// Se o estado de redundância deste PLC alterou...
IF NonRedData.bRedStateChanged THEN
	// Torna as saídas diferentes das entradas, garantindo que as consistências de dados
	// sejam feitas a partir de valores decorrentes de novas comunicações
	ATs.awModbus3HoldingWrite[0]:= ATs.awModbus3InputRegRead[0] + 100;
	// Inicializa temporizador para atrasar a consistência dos valores lidos, pois quando
	// o PLC assume como ativo, vai levar algum tempo até a comunicação ser estabelecida
	liAnalogTimer:= - ProjectConstants.iTimeToSkipAsActive;
ELSE
	// Se o protocolo MODBUS está rodando e se os dados são consistentes...
	IF DG_MODBUS_Client_3.tDiag.bRunning AND bStatusHolding AND bStatusInputReg THEN
		// Incrementa o valor escrito nos holding registers
		ATs.awModbus3HoldingWrite[0]:= ATs.awModbus3HoldingWrite[0] + 100;
		// Reseta o temporizador
		liAnalogTimer:= 0;
	ELSE
		// Acumula o tempo que passou
		liAnalogTimer:= liAnalogTimer + ProjectConstants.iMainTaskInterval;
		// Registra o tempo máximo
		MinMaxTimes.liAnaMaxTime_CheckModbus3:= MAX(MinMaxTimes.liAnaMaxTime_CheckModbus3, liAnalogTimer);
		// Caso o tempo máximo tenha sido extrapolado...
		IF liAnalogTimer >= ProjectConstants.iModbus3ReadWriteDelay THEN
			// Restarta o MODBUS caso o bug 17184 se manifeste.
			IF DG_MODBUS_Server_3.tStat.wActiveConnections = 0 THEN
				///DG_MODBUS_Server_3.tCommand.bRestart:= TRUE;
				PersistentVars.iBug17184_Counter_MDBUS3:= PersistentVars.iBug17184_Counter_MDBUS3 + 1;
				///iAnalogTimer:= - ProjectConstants.iTimeToSkipAsActive;
			ELSE	
				// Registra falha nos holding register, caso tenha ocorrido
				IF bStatusHolding = FALSE THEN
					PersistentVars.bModbus3ErrorHolding:= TRUE;
					awHoldingError_DataWr:= ATs.awModbus3HoldingWrite;
					awHoldingError_DataRd:= ATs.awModbus3HoldingRead;
				END_IF
				// Registra falha nos input register, caso tenha ocorrido
				IF bStatusInputReg = FALSE THEN
					PersistentVars.bModbus3ErrorInputReg:= TRUE;
					awInputRegError_DataWr:= ATs.awModbus3HoldingWrite;
					awInputRegError_DataRd:= ATs.awModbus3InputRegRead;
				END_IF
			END_IF
		END_IF
	END_IF
END_IF

// Atualiza os valores escritos
FOR wIndex:= 1 TO 119 BY 1 DO
	ATs.awModbus3HoldingWrite[wIndex]:= ATs.awModbus3HoldingWrite[wIndex - 1] + wIndex;
END_FOR

//
// Calcula a taxa média de comunicação
//

// Incrementa o número de milisegundos que transcorreram
iMilisecondsCounter:= iMilisecondsCounter + ProjectConstants.iMainTaskInterval;
// Se já se passou o tempo configurado desde a última média realizada...
IF iMilisecondsCounter >= ProjectConstants.iMsToComputeComRate THEN
	// Só calcula se o contador não virou
	IF DG_MODBUS_Client_3.tStat.wRXNormalResponses > wOldRXNormalResponses THEN
		// Calcula a taxa de comunicação atual
		MinMaxTimes.diModbus3BytesPerSec:=	WORD_TO_DINT(DG_MODBUS_Client_3.tStat.wRXNormalResponses - wOldRXNormalResponses) *
											iBytesPerResponse * 1000 / iMilisecondsCounter;
	END_IF
	// Zera o número de milisegundos transcorridos
	iMilisecondsCounter:= 0;
	// Salva número de respostas atuais
	wOldRXNormalResponses:= DG_MODBUS_Client_3.tStat.wRXNormalResponses;
END_IF

// Registra o tempo do sistema
SysTimeGetUs(uliPouEndTime);
// Calcula duração mínima/máxima desta POU
MinMaxTimes.uliPouMinTime_CheckModbus3:= MIN(MinMaxTimes.uliPouMinTime_CheckModbus3, uliPouEndTime - uliPouIniTime);
MinMaxTimes.uliPouMaxTime_CheckModbus3:= MAX(MinMaxTimes.uliPouMaxTime_CheckModbus3, uliPouEndTime - uliPouIniTime);

END_PROGRAM

// Device/Application/UserPOUs/Non-Redundant/CheckModbus4
PROGRAM CheckModbus4
VAR
	wIndex : WORD;
	bStatusCoil : BOOL;
	bStatusStatus : BOOL;
	bStatusHolding : BOOL;
	bStatusInputReg : BOOL;
	liDigitalTimer : LINT := 0;
	liAnalogTimer : LINT := 0;
	abCoilsError_DataWr : ARRAY [0..1919] OF BOOL;
	abCoilsError_DataRd : ARRAY [0..1919] OF BOOL;
	abStatusError_DataWr : ARRAY [0..1919] OF BOOL;
	abStatusError_DataRd : ARRAY [0..1919] OF BOOL;
	awHoldingError_DataWr : ARRAY [0..119] OF WORD;
	awHoldingError_DataRd : ARRAY [0..119] OF WORD;
	awInputRegError_DataWr : ARRAY [0..119] OF WORD;
	awInputRegError_DataRd : ARRAY [0..119] OF WORD;
	wOldRXNormalResponses : WORD;
	iMilisecondsCounter : INT;
	iBytesPerResponse : INT := 240;
	uliPouIniTime : ULINT;
	uliPouEndTime : ULINT;
END_VAR

// Consistencia da integridade dos dados trocados via MODBUS

// Registra o tempo do sistema
SysTimeGetUs(uliPouIniTime);

//
// Controle e consistência dos coils e input status
//

// Consiste os valores lidos
bStatusCoil:= TRUE;
bStatusStatus:= TRUE;
FOR wIndex:= 0 TO 1919 BY 1 DO
	bStatusCoil:= bStatusCoil AND (ModbusSymbol.abModbus4CoilsRead[wIndex] = ModbusSymbol.abModbus4CoilsWrite[wIndex]);
	bStatusStatus:= bStatusStatus AND (ModbusSymbol.abModbus4StatusRead[wIndex] = ModbusSymbol.abModbus4CoilsWrite[wIndex]);
END_FOR

// Se o estado de redundância deste PLC alterou...
IF NonRedData.bRedStateChanged THEN
	// Torna as saídas diferentes das entradas, garantindo que as consistências de dados
	// sejam feitas a partir de valores decorrentes de novas comunicações
	ModbusSymbol.abModbus4CoilsWrite[0]:= NOT ModbusSymbol.abModbus4StatusRead[0];
	// Inicializa temporizador para atrasar a consistência dos valores lidos, pois quando
	// o PLC assume como ativo, vai levar algum tempo até a comunicação ser estabelecida
	liDigitalTimer:= - ProjectConstants.iTimeToSkipAsActive;
ELSE
	// Se o protocolo MODBUS está rodando e se os dados são consistentes...
	IF DG_MODBUS_Client_4.tDiag.bRunning AND bStatusCoil AND bStatusStatus THEN
		// Complementa o valor dos coils
		ModbusSymbol.abModbus4CoilsWrite[0]:= NOT ModbusSymbol.abModbus4CoilsWrite[0];
		// Reseta o temporizador
		liDigitalTimer:= 0;
	ELSE
		// Acumula o tempo que passou
		liDigitalTimer:= liDigitalTimer + ProjectConstants.iMainTaskInterval;
		// Registra o tempo máximo
		MinMaxTimes.liDigMaxTime_CheckModbus4:= MAX(MinMaxTimes.liDigMaxTime_CheckModbus4, liDigitalTimer);
		// Caso o tempo máximo tenha sido extrapolado...
		IF liDigitalTimer >= ProjectConstants.iModbus4ReadWriteDelay THEN
		// Restarta o MODBUS caso o bug 17184 se manifeste.
			IF DG_MODBUS_Server_4.tStat.wActiveConnections = 0 THEN
				///DG_MODBUS_Server_4.tCommand.bRestart:= TRUE;
				PersistentVars.iBug17184_CounterDig_MDBUS4:= PersistentVars.iBug17184_CounterDig_MDBUS4 + 1;
				///iDigitalTimer:= - ProjectConstants.iTimeToSkipAsActive;
			ELSE
				// Registra falha nos coils, caso tenha ocorrido
				IF bStatusCoil = FALSE THEN
					PersistentVars.bModbus4ErrorCoil:= TRUE;
					abCoilsError_DataWr:= ModbusSymbol.abModbus4CoilsWrite;
					abCoilsError_DataRd:= ModbusSymbol.abModbus4CoilsRead;
				END_IF
				// Registra falha nos inputs, caso tenha ocorrido
				IF bStatusStatus = FALSE THEN
					PersistentVars.bModbus4ErrorStatus:= TRUE;
					abStatusError_DataWr:= ModbusSymbol.abModbus4CoilsWrite;
					abStatusError_DataRd:= ModbusSymbol.abModbus4StatusRead;
				END_IF
			END_IF
		END_IF
	END_IF
END_IF

// Atualiza os valores escritos
FOR wIndex:= 1 TO 1919 BY 1 DO
	ModbusSymbol.abModbus4CoilsWrite[wIndex]:= NOT ModbusSymbol.abModbus4CoilsWrite[wIndex - 1];
END_FOR

//
// Controle e consistência dos holding registers
//

// Consiste os valores lidos
bStatusHolding:= TRUE;
bStatusInputReg:= TRUE;
FOR wIndex:= 0 TO 119 BY 1 DO
	bStatusHolding:= bStatusHolding AND (ModbusSymbol.awModbus4HoldingRead[wIndex] = ModbusSymbol.awModbus4HoldingWrite[wIndex]);
	bStatusInputReg:= bStatusInputReg AND (ModbusSymbol.awModbus4InputRegRead[wIndex] = ModbusSymbol.awModbus4HoldingWrite[wIndex]);
END_FOR

// Se o estado de redundância deste PLC alterou...
IF NonRedData.bRedStateChanged THEN
	// Torna as saídas diferentes das entradas, garantindo que as consistências de dados
	// sejam feitas a partir de valores decorrentes de novas comunicações
	ModbusSymbol.awModbus4HoldingWrite[0]:= ModbusSymbol.awModbus4InputRegRead[0] + 100;
	// Inicializa temporizador para atrasar a consistência dos valores lidos, pois quando
	// o PLC assume como ativo, vai levar algum tempo até a comunicação ser estabelecida
	liAnalogTimer:= - ProjectConstants.iTimeToSkipAsActive;
ELSE
	// Se o protocolo MODBUS está rodando e se os dados são consistentes...
	IF DG_MODBUS_Client_4.tDiag.bRunning AND bStatusHolding AND bStatusInputReg THEN
		// Incrementa o valor escrito nos holding registers
		ModbusSymbol.awModbus4HoldingWrite[0]:= ModbusSymbol.awModbus4HoldingWrite[0] + 100;
		// Reseta o temporizador
		liAnalogTimer:= 0;
	ELSE
		// Acumula o tempo que passou
		liAnalogTimer:= liAnalogTimer + ProjectConstants.iMainTaskInterval;
		// Registra o tempo máximo
		MinMaxTimes.liAnaMaxTime_CheckModbus4:= MAX(MinMaxTimes.liAnaMaxTime_CheckModbus4, liAnalogTimer);
		// Caso o tempo máximo tenha sido extrapolado...
		IF liAnalogTimer >= ProjectConstants.iModbus4ReadWriteDelay THEN
			// Restarta o MODBUS caso o bug 17184 se manifeste.
			IF DG_MODBUS_Server_4.tStat.wActiveConnections = 0 THEN
				///DG_MODBUS_Server_4.tCommand.bRestart:= TRUE;
				PersistentVars.iBug17184_Counter_MDBUS4:= PersistentVars.iBug17184_Counter_MDBUS4 + 1;
				///AnalogTimer:= - ProjectConstants.iTimeToSkipAsActive;
			ELSE
				// Registra falha nos holding register, caso tenha ocorrido
				IF bStatusHolding = FALSE THEN
					PersistentVars.bModbus4ErrorHolding:= TRUE;
					awHoldingError_DataWr:= ModbusSymbol.awModbus4HoldingWrite;
					awHoldingError_DataRd:= ModbusSymbol.awModbus4HoldingRead;
				END_IF
				// Registra falha nos input register, caso tenha ocorrido
				IF bStatusInputReg = FALSE THEN
					PersistentVars.bModbus4ErrorInputReg:= TRUE;
					awInputRegError_DataWr:= ModbusSymbol.awModbus4HoldingWrite;
					awInputRegError_DataRd:= ModbusSymbol.awModbus4InputRegRead;
				END_IF
			END_IF
		END_IF
	END_IF
END_IF

// Atualiza os valores escritos
FOR wIndex:= 1 TO 119 BY 1 DO
	ModbusSymbol.awModbus4HoldingWrite[wIndex]:= ModbusSymbol.awModbus4HoldingWrite[wIndex - 1] + wIndex;
END_FOR

//
// Calcula a taxa média de comunicação
//

// Incrementa o número de milisegundos que transcorreram
iMilisecondsCounter:= iMilisecondsCounter + ProjectConstants.iMainTaskInterval;
// Se já se passou o tempo configurado desde a última média realizada...
IF iMilisecondsCounter >= ProjectConstants.iMsToComputeComRate THEN
	// Só calcula se o contador não virou
	IF DG_MODBUS_Client_4.tStat.wRXNormalResponses > wOldRXNormalResponses THEN
		// Calcula a taxa de comunicação atual
		MinMaxTimes.diModbus4BytesPerSec:=	WORD_TO_DINT(DG_MODBUS_Client_4.tStat.wRXNormalResponses - wOldRXNormalResponses) *
											iBytesPerResponse * 1000 / iMilisecondsCounter;
	END_IF
	// Zera o número de milisegundos transcorridos
	iMilisecondsCounter:= 0;
	// Salva número de respostas atuais
	wOldRXNormalResponses:= DG_MODBUS_Client_4.tStat.wRXNormalResponses;
END_IF

// Registra o tempo do sistema
SysTimeGetUs(uliPouEndTime);
// Calcula duração mínima/máxima desta POU
MinMaxTimes.uliPouMinTime_CheckModbus4:= MIN(MinMaxTimes.uliPouMinTime_CheckModbus4, uliPouEndTime - uliPouIniTime);
MinMaxTimes.uliPouMaxTime_CheckModbus4:= MAX(MinMaxTimes.uliPouMaxTime_CheckModbus4, uliPouEndTime - uliPouIniTime);

END_PROGRAM

// Device/Application/UserPOUs/Redundant/CheckProfibusIOs
PROGRAM CheckProfibusIOs
VAR
	iAnalogHigh : INT := 30000;
	iAnalogLow : INT := 1500;
	iAnalogError : INT := 100;
	iAnalogStep : INT := 1500;
	abErrorLoopBack : ARRAY [0..3] OF BYTE;
	uliPouIniTime : ULINT;
	uliPouEndTime : ULINT;
END_VAR

// Registra o tempo do sistema
SysTimeGetUs(uliPouIniTime);

// Zera variáveis em caso de comando para reinicializar os contadores de diagnóstico
	IF Symbolics.bEnableCleanStats_CheckProfibusIOs = TRUE THEN
		abErrorLoopBack[0]:= 0;
		abErrorLoopBack[1]:= 0;
		abErrorLoopBack[2]:= 0;
		abErrorLoopBack[3]:= 0;
		Symbolics.bEnableCleanStats_CheckProfibusIOs:= FALSE;
	END_IF



//
// Teste de consistência de I/Os PROFIBUS digitais e analógicos ligados ao PO5065.
//

// Se o mestre Profibus está presente no barramento e se a primeira cabeça (endereço 5) está ativa na rede...
IF (((DG_NX3030.tDetailed.WHSB.adwModulePresenceStatus[0] AND 2#001000000) > 0) AND
	 (DG_NX5001_1.tRedund.tActivNtw.bSlave_5 = TRUE)) OR
   (((DG_NX3030.tDetailed.WHSB.adwModulePresenceStatus[0] AND 2#100000000) > 0) AND
	 (DG_NX5001_2.tRedund.tActivNtw.bSlave_5 = TRUE)) THEN
	// Se os módulos de entrada e de saída digital estiverem presentes no barramento...
	IF (DG_PO5065_05.tPbusHeadA.tModule_0to7_Status.bModuleNotFound_00 = FALSE) AND
	   (DG_PO5065_05.tPbusHeadA.tModule_0to7_Status.bModuleNotFound_01 = FALSE) AND
	   (DG_PO5065_05.tPbusHeadB.tModule_0to7_Status.bModuleNotFound_00 = FALSE) AND 
	   (DG_PO5065_05.tPbusHeadB.tModule_0to7_Status.bModuleNotFound_01 = FALSE) THEN
		// Consiste entradas e saídas digitais, interligadas fisicamente
		IF REM05_PO2020_G0 = REM05_PO1000_G0 THEN
			// Incrementa o estado das saídas digitais
			REM05_PO2020_G0:= REM05_PO2020_G0 + 1;
			// Reseta o temporizador
			NonRedData.iProfibus5DigTimer:= 0;
		ELSE
			// Acumula o tempo que passou
			NonRedData.iProfibus5DigTimer:= NonRedData.iProfibus5DigTimer + ProjectConstants.iMainTaskInterval;
			// Registra o tempo máximo
			MinMaxTimes.liDigMaxTime_CheckProfibusIOs:= MAX(MinMaxTimes.liDigMaxTime_CheckProfibusIOs, NonRedData.iProfibus5DigTimer);
			// Aguarda a passagem do tempo antes de considerar falha
			IF NonRedData.iProfibus5DigTimer = ProjectConstants.iProfibusDelayDigital THEN
				// Contabiliza erro de consistência dos pontos digitais
				PersistentVars.dwSlave5DigIOsErrors:= PersistentVars.dwSlave5DigIOsErrors + 1;
				//Armazena o erro da entrada e saida
				abErrorLoopBack[0]:= REM05_PO1000_G0;
				abErrorLoopBack[1]:= REM05_PO2020_G0;
			ELSE
				//Gabriel Fonseca - 28/10/2022
				//Verifica se congelou por mais de um ciclo, retornar >= no if acima 
				IF NonRedData.iProfibus5DigTimer >= 2* ProjectConstants.iProfibusDelayDigital THEN
					PersistentVars.bFrozenErrorRem05TORem05:= TRUE;
				END_IF
			END_IF
		END_IF
	// Se algum dos módulos de entrada e de saída digital estiverem ausentes do barramento...
	ELSE
		// Acumula o tempo que passou
		NonRedData.iProfibus5DigTimer:= NonRedData.iProfibus5DigTimer + ProjectConstants.iMainTaskInterval;
		// Registra o tempo máximo
		MinMaxTimes.liDigMaxTime_CheckProfibusIOs:= MAX(MinMaxTimes.liDigMaxTime_CheckProfibusIOs, NonRedData.iProfibus5DigTimer);
		// Aguarda a passagem do tempo antes de considerar falha
		IF NonRedData.iProfibus5DigTimer >= ProjectConstants.iProfibusDelayDigital THEN
			// Contabiliza erro de módulo ausente do barramento
			PersistentVars.dwSlave5ModulesOut:= PersistentVars.dwSlave5ModulesOut + 1;
		END_IF
	END_IF
// Se o mestre Profibus está ausente do barramento ou se a primeira cabeça (endereço 5) não está ativa na rede...
ELSE
	// Acumula o tempo que passou
	NonRedData.iProfibus5DigTimer:= NonRedData.iProfibus5DigTimer + ProjectConstants.iMainTaskInterval;
	// Registra o tempo máximo
	MinMaxTimes.liDigMaxTime_CheckProfibusIOs:= MAX(MinMaxTimes.liDigMaxTime_CheckProfibusIOs, NonRedData.iProfibus5DigTimer);
	// Aguarda a passagem do tempo antes de considerar falha
	IF NonRedData.iProfibus5DigTimer >= ProjectConstants.iProfibusDelayDigital THEN
		// Contabiliza erro de Cabeça não ativa na rede
		PersistentVars.dwSlave5Unavailable:= PersistentVars.dwSlave5Unavailable + 1;
	END_IF
END_IF

// Se o mestre Profibus está presente no barramento e se a segunda cabeça (endereço 10) está ativa na rede...
IF (((DG_NX3030.tDetailed.WHSB.adwModulePresenceStatus[0] AND 2#001000000) > 0) AND 
	 (DG_NX5001_1.tRedund.tActivNtw.bSlave_10 = TRUE)) OR
   (((DG_NX3030.tDetailed.WHSB.adwModulePresenceStatus[0] AND 2#100000000) > 0) AND 
	 (DG_NX5001_2.tRedund.tActivNtw.bSlave_10 = TRUE)) THEN
	// Se os módulos de entrada e de saída analógica estiverem presentes no barramento...
	IF (DG_PO5065_10.tPbusHeadA.tModule_0to7_Status.bModuleNotFound_00 = FALSE) AND
	   (DG_PO5065_10.tPbusHeadA.tModule_0to7_Status.bModuleNotFound_01 = FALSE) AND
	   (DG_PO5065_10.tPbusHeadB.tModule_0to7_Status.bModuleNotFound_00 = FALSE) AND
	   (DG_PO5065_10.tPbusHeadB.tModule_0to7_Status.bModuleNotFound_01 = FALSE) THEN
		// Consistência da primeira entrada analógica (rampa)
		IF (WORD_TO_INT(REM10_PO1212_C00) >= (Symbolics.iAnalogValue - iAnalogError)) AND
		   (WORD_TO_INT(REM10_PO1212_C00) <= (Symbolics.iAnalogValue + iAnalogError)) THEN
			// Implementa rampa analógica
			Symbolics.iAnalogValue:= Symbolics.iAnalogValue + iAnalogStep;
			// Ajusta subida/descida da rampa analógica
			IF Symbolics.iAnalogValue >= iAnalogHigh THEN
				Symbolics.iAnalogValue:= iAnalogHigh;
				iAnalogStep:= -iAnalogStep;
			END_IF
			IF Symbolics.iAnalogValue <= iAnalogLow	THEN
				Symbolics.iAnalogValue:= iAnalogLow;
				iAnalogStep:= -iAnalogStep;
			END_IF
			// Primeira saída analógica é uma rampa
			REM10_PO2132_C00:= INT_TO_WORD(Symbolics.iAnalogValue);
			// Reseta o temporizador
			NonRedData.iProfibus10AnaTimer:= 0;
		ELSE
			// Acumula o tempo que passou
			NonRedData.iProfibus10AnaTimer:= NonRedData.iProfibus10AnaTimer + ProjectConstants.iMainTaskInterval;
			// Registra o tempo máximo
			MinMaxTimes.liAnaMaxTime_CheckProfibusIOs:= MAX(MinMaxTimes.liAnaMaxTime_CheckProfibusIOs, NonRedData.iProfibus10AnaTimer);
			// Aguarda a passagem do tempo antes de considerar falha
			IF NonRedData.iProfibus10AnaTimer >= ProjectConstants.iProfibusDelayAnalog THEN
				// Contabiliza erro de consistência dos pontos analógicos
				PersistentVars.dwSlave10AnaIOsErrors:= PersistentVars.dwSlave10AnaIOsErrors + 1;
				// Salva os valores errados
				PersistentVars.wErrorValuePO2132C00:= REM10_PO2132_C00;
				PersistentVars.wErrorValuePO1212C00:= REM10_PO1212_C00;
			END_IF
		END_IF
	// Se algum dos módulos de entrada e de saída analógica estiverem ausentes do barramento...
	ELSE
		// Acumula o tempo que passou
		NonRedData.iProfibus10AnaTimer:= NonRedData.iProfibus10AnaTimer + ProjectConstants.iMainTaskInterval;
		// Registra o tempo máximo
		MinMaxTimes.liAnaMaxTime_CheckProfibusIOs:= MAX(MinMaxTimes.liAnaMaxTime_CheckProfibusIOs, NonRedData.iProfibus10AnaTimer);
		// Aguarda a passagem do tempo antes de considerar falha
		IF NonRedData.iProfibus10AnaTimer >= ProjectConstants.iProfibusDelayAnalog THEN
			// Contabiliza erro de módulo ausente do barramento
			PersistentVars.dwSlave10ModulesOut:= PersistentVars.dwSlave10ModulesOut + 1;
		END_IF
	END_IF
// Se o mestre Profibus está ausente do barramento ou se a segunda cabeça (endereço 10) não está ativa na rede...
ELSE
	// Acumula o tempo que passou
	NonRedData.iProfibus10AnaTimer:= NonRedData.iProfibus10AnaTimer + ProjectConstants.iMainTaskInterval;
	// Registra o tempo máximo
	MinMaxTimes.liAnaMaxTime_CheckProfibusIOs:= MAX(MinMaxTimes.liAnaMaxTime_CheckProfibusIOs, NonRedData.iProfibus10AnaTimer);
	// Aguarda a passagem do tempo antes de considerar falha
	IF NonRedData.iProfibus10AnaTimer >= ProjectConstants.iProfibusDelayAnalog THEN
		// Contabiliza erro de Cabeça não ativa na rede
		PersistentVars.dwSlave10Unavailable:= PersistentVars.dwSlave10Unavailable + 1;
	END_IF
END_IF

//
// Teste de consistência de I/Os PROFIBUS digital ligado ao PO5063.
//

// Se o mestre Profibus está presente no barramento e se a cabeça (endereço 3) está ativa na rede...
IF (((DG_NX3030.tDetailed.WHSB.adwModulePresenceStatus[0] AND 2#10000000000000000) > 0) AND //posição 16
	 (DG_NX5001_3.tMstStatus.abySlv_State.bSlave_4 = TRUE)) THEN
	// Se o módulo de entrada digital estiver presente no barramento...
	IF DG_PO5063_04.tPbusHeadA.tModule_0to7_Status.bModuleNotFound_00 = FALSE THEN
		// Consiste entradas e saídas digitais, interligadas fisicamente
		
		IF REM05_PO2020_G1 = REM04_PO1000_G0 THEN
			// Incrementa o estado das saídas digitais
			REM05_PO2020_G1:= REM05_PO2020_G1 + 1;
			// Reseta o temporizador
			NonRedData.iProfibus3DigTimer:= 0;
		ELSE
			// Acumula o tempo que passou
			NonRedData.iProfibus3DigTimer:= NonRedData.iProfibus3DigTimer + ProjectConstants.iMainTaskInterval;
			// Registra o tempo máximo
			MinMaxTimes.liDigMaxTime_CheckProfibusIOs:= MAX(MinMaxTimes.liDigMaxTime_CheckProfibusIOs, NonRedData.iProfibus3DigTimer);
			// Aguarda a passagem do tempo antes de considerar falha
			IF NonRedData.iProfibus3DigTimer = ProjectConstants.iProfibusDelayDigital THEN
				// Contabiliza erro de consistência dos pontos digitais
				PersistentVars.dwSlave3DigIOsErrors:= PersistentVars.dwSlave3DigIOsErrors + 1;
				//Armazena o erro da entrada e saida
				abErrorLoopBack[2] := REM04_PO1000_G0;
				abErrorLoopBack[3] := REM05_PO2020_G1;
			ELSE 
				//Gabriel Fonseca - 28/10/2022
				//Verifica se congelou por mais de um ciclo, retornar >= no if acima 
				IF NonRedData.iProfibus3DigTimer >= 2* ProjectConstants.iProfibusDelayDigital THEN
					PersistentVars.bFrozenErrorRem05TORem04:= TRUE;
				END_IF
			END_IF
			
		END_IF
	// Se o módulo de entrada digital estiver ausente do barramento...
	ELSE
		// Acumula o tempo que passou
		NonRedData.iProfibus3DigTimer:= NonRedData.iProfibus3DigTimer + ProjectConstants.iMainTaskInterval;
		// Registra o tempo máximo
		MinMaxTimes.liDigMaxTime_CheckProfibusIOs:= MAX(MinMaxTimes.liDigMaxTime_CheckProfibusIOs, NonRedData.iProfibus3DigTimer);
		// Aguarda a passagem do tempo antes de considerar falha
		IF NonRedData.iProfibus3DigTimer >= ProjectConstants.iProfibusDelayDigital THEN
			// Contabiliza erro de módulo ausente do barramento
			PersistentVars.dwSlave3ModulesOut:= PersistentVars.dwSlave3ModulesOut + 1;
		END_IF
	END_IF
// Se o mestre Profibus está ausente do barramento ou se a cabeça (endereço 3) não está ativa na rede...
ELSE
	// Acumula o tempo que passou
	NonRedData.iProfibus3DigTimer:= NonRedData.iProfibus3DigTimer + ProjectConstants.iMainTaskInterval;
	// Registra o tempo máximo
	MinMaxTimes.liDigMaxTime_CheckProfibusIOs:= MAX(MinMaxTimes.liDigMaxTime_CheckProfibusIOs, NonRedData.iProfibus3DigTimer);
	// Aguarda a passagem do tempo antes de considerar falha
	IF NonRedData.iProfibus3DigTimer >= ProjectConstants.iProfibusDelayDigital THEN
		// Contabiliza erro de Cabeça não ativa na rede
		PersistentVars.dwSlave3Unavailable:= PersistentVars.dwSlave3Unavailable + 1;
	END_IF
END_IF

//*****************************************************************************************************************************************************************************
//
// Teste de consistência de I/Os PROFIBUS ligados a remotas Nexto

// Registra o tempo do sistema
SysTimeGetUs(uliPouEndTime);
// Calcula duração mínima/máxima desta POU
MinMaxTimes.uliPouMinTime_CheckProfibusIOs:= MIN(MinMaxTimes.uliPouMinTime_CheckProfibusIOs, uliPouEndTime - uliPouIniTime);
MinMaxTimes.uliPouMaxTime_CheckProfibusIOs:= MAX(MinMaxTimes.uliPouMaxTime_CheckProfibusIOs, uliPouEndTime - uliPouIniTime);

END_PROGRAM

// Device/Application/UserPOUs/Redundant/CheckRecipe
PROGRAM CheckRecipe
VAR
	sName : STRING := 'ReceitaMinima';
	sDef : STRING := 'Machine01';
	mRET : RECIPE_RETURN_VALUES;
	boolStartProcess : BOOL;
	bTestRecipe : BOOL;
	iCounterCycle : INT;
	bOneCycle : BOOL;
	uliPouIniTime : ULINT;
	uliPouEndTime : ULINT;
END_VAR

//*****************************************************************************
// Autor(es): Roberto Martiny
// Descrição:
// Esta POU testa a funcionalidade do Recipe Manager.
//*****************************************************************************

// Registra o tempo do sistema
SysTimeGetUs(uliPouIniTime);

//*****************************************************************************
// Testa Recipe Manager

IF bOneCycle = FALSE THEN
	mRET := WriteRecipe(SDef,SName);
	bOneCycle := TRUE;
END_IF

iCounterCycle := iCounterCycle+1;

IF bTestRecipe = FALSE AND iCounterCycle > 1 THEN
	IF Recipe.iRecipeValueA <> -1000 OR Recipe.iRecipeValueB <> 1 OR Recipe.iRecipeValueC <> -900 THEN
	PersistentVars.dwRecipeErrors := PersistentVars.dwRecipeErrors +1;
	END_IF
	// fica por 10 ciclos consistindo este recipe
	IF iCounterCycle > 10 THEN
		iCounterCycle :=0;
		bTestRecipe := TRUE;
		sName := 'ReceitaMaxima';
		mRET := WriteRecipe(SDef,SName);	
	END_IF	
END_IF

IF bTestRecipe = TRUE  AND iCounterCycle > 1 THEN
	IF Recipe.iRecipeValueA <> 1000 OR Recipe.iRecipeValueB <> 900 OR Recipe.iRecipeValueC <> -1 THEN
	PersistentVars.dwRecipeErrors := PersistentVars.dwRecipeErrors +1;
	END_IF
	// fica por 10 ciclos consistindo este recipe
	IF iCounterCycle > 10 THEN
		iCounterCycle :=0;
		bTestRecipe := FALSE;
		sName := 'ReceitaMinima';
		mRET := WriteRecipe(SDef,SName);
	END_IF	
END_IF

// Verifica retorno da função de escrita do Recipe
IF mRET <> RECIPE_RETURN_VALUES.ERROR_OK THEN
	PersistentVars.dwRecipeReturnError := mRET;
END_IF;
//*****************************************************************************

// Registra o tempo do sistema
SysTimeGetUs(uliPouEndTime);
// Calcula duração mínima/máxima desta POU
MinMaxTimes.uliPouMinTime_CheckRecipe:= MIN(MinMaxTimes.uliPouMinTime_CheckRecipe, uliPouEndTime - uliPouIniTime);
MinMaxTimes.uliPouMaxTime_CheckRecipe:= MAX(MinMaxTimes.uliPouMaxTime_CheckRecipe, uliPouEndTime - uliPouIniTime);

END_PROGRAM

// Device/Application/UserPOUs/Redundant/CheckSoe
PROGRAM CheckSoe
VAR
	wCounter : WORD := 0;
	wOldCounter : WORD := 0;
	// Memórias de salvamento dos erros
	wMemError_Soe1OverflowOldCounter : WORD;
	wMemError_Soe2OverflowOldCounter : WORD;
	wMemError_Soe1Diagnostic : WORD;
	wMemError_Soe1OldCounter : WORD;
	wMemError_Soe2Diagnostic : WORD;
	wMemError_Soe2OldCounter : WORD;
	uliPouIniTime : ULINT;
	uliPouEndTime : ULINT;
END_VAR

// Gera dois eventos SOE a cada ciclo nos dois servers e consiste a existência dos mesmos na fila.

// Registra o tempo do sistema
SysTimeGetUs(uliPouIniTime);

// Retorna se for o primeiro ciclo como ativo, pois os diagnósticos não estão atualizados
// Retorna também se for o segundo ciclo como ativo, devido ao BUG 17134
IF NonRedData.aeLastRedState[1] <> REDUNDANCY_STATE.ACTIVE OR
   NonRedData.aeLastRedState[2] <> REDUNDANCY_STATE.ACTIVE THEN
	RETURN;
END_IF

// Se for a primeira vez que esta POU será executada como PLC ativo, deve considerar a
// quantidade de eventos que já estão na fila, inclusive o overflow, pois são retentivos
IF NonRedData.bSoeFirstCheckCycle = TRUE THEN
	wCounter:= wOldCounter:= DG_NX3030.tDetailed.SOE[1].wEventsCounter +
							 2 * BOOL_TO_WORD(DG_NX3030.tDetailed.SOE[1].bOverflowStatus);
	NonRedData.bSoeFirstCheckCycle:= FALSE;
END_IF

//
// Consistência da indicação de overflow
//

// Se já ultrapassou o limite de eventos suportado, deve ter ligado o overflow
IF wOldCounter > ProjectConstants.wSoeEventQueueSize THEN
	// Se o flag de overflow da fila 1 está desligado...
	IF DG_NX3030.tDetailed.SOE[1].bOverflowStatus = FALSE THEN
		// Indica a ocorrência de um falso overflow
		PersistentVars.bSOE1FalseOverflow:= TRUE;
		// Salva os valores nas memórias de erro
		wMemError_Soe1OverflowOldCounter:= wOldCounter;
	END_IF
	// Se o flag de overflow da fila 2 está desligado...
	IF DG_NX3030.tDetailed.SOE[2].bOverflowStatus = FALSE THEN
		// Indica a ocorrência de um falso overflow
		PersistentVars.bSOE2FalseOverflow:= TRUE;
		// Salva os valores nas memórias de erro
		wMemError_Soe2OverflowOldCounter:= wOldCounter;
	END_IF
// Se não ultrapassou o limite de eventos suportado, não deve ter ligado o overflow
ELSE
	// Se o flag de overflow da fila 1 está ligado...
	IF DG_NX3030.tDetailed.SOE[1].bOverflowStatus = TRUE THEN
		// Indica a ocorrência de um falso overflow
		PersistentVars.bSOE1FalseOverflow:= TRUE;
		// Salva os valores nas memórias de erro
		wMemError_Soe1OverflowOldCounter:= wOldCounter;
	END_IF
	// Se o flag de overflow da fila 2 está ligado...
	IF DG_NX3030.tDetailed.SOE[2].bOverflowStatus = TRUE THEN
		// Indica a ocorrência de um falso overflow
		PersistentVars.bSOE2FalseOverflow:= TRUE;
		// Salva os valores nas memórias de erro
		wMemError_Soe2OverflowOldCounter:= wOldCounter;
	END_IF
END_IF

//
// Consistência da quantidade de eventos gerados
//

// Se não ultrapassou o limite de eventos suportado pela fila...
IF wOldCounter <= ProjectConstants.wSoeEventQueueSize THEN
	// Se o número de eventos na fila 1 não confere com o número de eventos gerados...
	IF DG_NX3030.tDetailed.SOE[1].wEventsCounter <> wOldCounter THEN
		// Indica falha na quantidade de eventos
		PersistentVars.bSOE1EventsMismatch:= TRUE;
		// Salva os valores nas memórias de erro
		wMemError_Soe1Diagnostic:= DG_NX3030.tDetailed.SOE[1].wEventsCounter;
		wMemError_Soe1OldCounter:= wOldCounter;
	END_IF
	// Se o número de eventos na fila 2 não confere com o número de eventos gerados...
	IF DG_NX3030.tDetailed.SOE[2].wEventsCounter <> wOldCounter THEN
		// Indica falha na quantidade de eventos
		PersistentVars.bSOE2EventsMismatch:= TRUE;
		// Salva os valores nas memórias de erro
		wMemError_Soe2Diagnostic:= DG_NX3030.tDetailed.SOE[2].wEventsCounter;
		wMemError_Soe2OldCounter:= wOldCounter;
	END_IF
// Se já ultrapassou o limite de eventos suportado pela fila...
ELSE
	// Se o número de eventos na fila 1 não confere com o número máximo...
	IF DG_NX3030.tDetailed.SOE[1].wEventsCounter <> ProjectConstants.wSoeEventQueueSize THEN
		// Indica falha na quantidade de eventos
		PersistentVars.bSOE1EventsMismatch:= TRUE;
		// Salva os valores nas memórias de erro
		wMemError_Soe1Diagnostic:= DG_NX3030.tDetailed.SOE[1].wEventsCounter;
		wMemError_Soe1OldCounter:= wOldCounter;
	END_IF
	// Se o número de eventos na fila 2 não confere com o número máximo...
	IF DG_NX3030.tDetailed.SOE[2].wEventsCounter <> ProjectConstants.wSoeEventQueueSize THEN
		// Indica falha na quantidade de eventos
		PersistentVars.bSOE2EventsMismatch:= TRUE;
		// Salva os valores nas memórias de erro
		wMemError_Soe2Diagnostic:= DG_NX3030.tDetailed.SOE[2].wEventsCounter;
		wMemError_Soe2OldCounter:= wOldCounter;
	END_IF
END_IF

// Salva o contador atual para consistir no próximo ciclo. Isto é necessário pois
// os diagnósticos (por exemplo, de eventos na fila) estão defasados em um ciclo:
// ao final da MainPrg, primeiro são gerados os diagnósticos e depois os eventos.  
wOldCounter:= wCounter;

// Enquanto não atingir o limite, gera mais dois eventos por ciclo
IF wCounter < ANY_TO_WORD(wCounter + 2) THEN
	ATs.bSOEPoint000:= NOT(ATs.bSOEPoint000);
	ATs.bSOEPoint999:= NOT(ATs.bSOEPoint999);
	wCounter:= wCounter + 2;
// Código para manter a instrução IF simétrica
ELSE
	ATs.bSOEPoint000:= ATs.bSOEPoint000;
	ATs.bSOEPoint999:= ATs.bSOEPoint999;
	wCounter:= wCounter + 0;
END_IF

// Registra o tempo do sistema
SysTimeGetUs(uliPouEndTime);
// Calcula duração mínima/máxima desta POU
MinMaxTimes.uliPouMinTime_CheckSoe:= MIN(MinMaxTimes.uliPouMinTime_CheckSoe, uliPouEndTime - uliPouIniTime);
MinMaxTimes.uliPouMaxTime_CheckSoe:= MAX(MinMaxTimes.uliPouMaxTime_CheckSoe, uliPouEndTime - uliPouIniTime);

END_PROGRAM

// Device/Application/UserPOUs/Redundant/CheckLanguages
PROGRAM CheckLanguages
VAR
	idelayFirstSecond : INT;
	uliPouIniTime : ULINT;
	uliPouEndTime : ULINT;
END_VAR

// Esta POU testa todas as linguagens de programação.
// Está toda estruturada dentro da SFC.

// Registra o tempo do sistema
SysTimeGetUs(uliPouIniTime);

POU_SFC(); 
IF idelayFirstSecond > 5 THEN
	IF languages.bResultado_POU_SFC <> TRUE THEN
		Persistentvars.dwErrorLanguages := Persistentvars.dwErrorLanguages + 1;	
	END_IF
ELSE
	idelayFirstSecond := idelayFirstSecond + 1;
END_IF

// Registra o tempo do sistema
SysTimeGetUs(uliPouEndTime);
// Calcula duração mínima/máxima desta POU
MinMaxTimes.uliPouMinTime_CheckLanguages:= MIN(MinMaxTimes.uliPouMinTime_CheckLanguages, uliPouEndTime - uliPouIniTime);
MinMaxTimes.uliPouMaxTime_CheckLanguages:= MAX(MinMaxTimes.uliPouMaxTime_CheckLanguages, uliPouEndTime - uliPouIniTime);

END_PROGRAM

// Device/Application/UserPOUs/Redundant/Languages/POU_SFC
PROGRAM POU_SFC
VAR
	Resul_CFC: BOOL;
	Resul_IL: BOOL;
	Resul_FBD: BOOL;
	Resul_LD: BOOL;
END_VAR

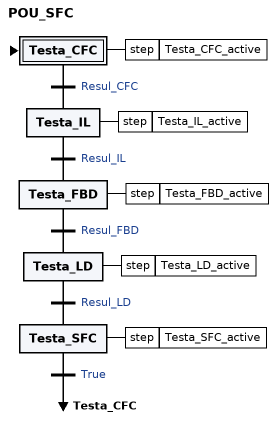
INITIAL_STEP Testa_CFC:
    Testa_CFC_active(N);  // step action
END_STEP
TRANSITION FROM Testa_CFC TO Testa_IL
    := Resul_CFC;
END_TRANSITION
STEP Testa_IL:
    Testa_IL_active(N);  // step action
END_STEP
TRANSITION FROM Testa_IL TO Testa_FBD
    := Resul_IL;
END_TRANSITION
STEP Testa_FBD:
    Testa_FBD_active(N);  // step action
END_STEP
TRANSITION FROM Testa_FBD TO Testa_LD
    := Resul_FBD;
END_TRANSITION
STEP Testa_LD:
    Testa_LD_active(N);  // step action
END_STEP
TRANSITION FROM Testa_LD TO Testa_SFC
    := Resul_LD;
END_TRANSITION
STEP Testa_SFC:
    Testa_SFC_active(N);  // step action
END_STEP
TRANSITION FROM Testa_SFC TO Testa_CFC
    := True;
END_TRANSITION

ACTION Testa_LD_active:
POU_LD();
IF languages.iResultado_POU_LD = 112 THEN
	Resul_LD:= TRUE;
END_IF
END_ACTION

ACTION Testa_IL_active:
POU_IL();
IF languages.iResultado_POU_IL = 118 THEN
	Resul_IL:= TRUE;
END_IF
END_ACTION

ACTION Testa_CFC_active:
POU_CFC();
POU_CFC_1000();
IF languages.iResultado_POU_CFC = 198 THEN
	Resul_CFC:= TRUE;
END_IF
END_ACTION

ACTION Testa_SFC_active:
Languages.bResultado_POU_SFC := TRUE;
END_ACTION

ACTION Testa_FBD_active:
POU_FBD();
IF languages.iResultado_POU_FBD = 112 THEN
	Resul_FBD:= TRUE;
END_IF
END_ACTION

END_PROGRAM

// Device/Application/UserPOUs/Redundant/Languages/POU_LD
PROGRAM POU_LD
VAR
// Variáveis para testar ADD de 2 entradas
	bHab01	: BOOL := FALSE;
	iSom01A	: INT :=1;
	iSom01B : INT :=2;
	iSom01R : INT; // valor esperado = 3
	
// Variáveis para testar ADD de 3 entradas
	bHab02	: BOOL := TRUE;
	iSom02A	: INT :=1;
	iSom02B : INT :=2;
	iSom02C : INT :=3;
	iSom02R : INT; // valor esperado = 6
	
// Variáveis para testar SUB de 2 entradas
	bHab03	: BOOL := TRUE;
	iSub03A	: INT :=3;
	iSub03B : INT :=2;
	iSub03R : INT; // valor esperado = 1
	
// Variáveis para testar MUL de 2 entradas
	bHab04	: BOOL := TRUE;
	iMul04A	: INT :=4;
	iMul04B : INT :=4;
	iMul04R : INT; // valor esperado = 16
	
// Variáveis para testar DIV de 2 entradas
	bHab05	: BOOL := TRUE;
	iDiv05A	: INT :=20;
	iDiv05B : INT :=5;
	iDiv05R : INT; // valor esperado = 4
	
// Variáveis para testar EQ de 2 entradas
	bHab06	: BOOL := FALSE;
	iEq06A	: INT :=25;
	iEq06B : INT :=25;
	bEq06R : BOOL; // valor esperado = true	

// Variáveis para testar NE de 2 entradas
	bHab07	: BOOL := TRUE;
	iNe07A	: INT :=24;
	iNe07B : INT :=25;
	bNe07R : BOOL; // valor esperado = true

// Variáveis para testar LT de 2 entradas
	bHab08	: BOOL := TRUE;
	iLt08A	: INT :=24;
	iLt08B : INT :=25;
	bLt08R : BOOL; // valor esperado = true		
	
// Variáveis para testar LE de 2 entradas
	bHab09	: BOOL := TRUE;
	iLe09A	: INT :=25;
	iLe09B : INT :=25;
	bLe09R : BOOL; // valor esperado = true		
	
// Variáveis para testar GT de 2 entradas
	bHab10	: BOOL := TRUE;
	iGt10A	: INT :=26;
	iGt10B : INT :=25;
	bGt10R : BOOL; // valor esperado = true	

// Variáveis para testar GE de 2 entradas
	bHab11	: BOOL := TRUE;
	iGe11A	: INT :=26;
	iGe11B : INT :=26;
	bGe11R : BOOL; // valor esperado = true		
	
// Variáveis para testar SEL
	bHab12	: BOOL := TRUE;
	bSelG : BOOL := TRUE;
	iSel12A	: INT :=20;
	iSel12B : INT :=26;
	iSel12R : INT; // valor esperado = 26		
	
// Variáveis para testar MUX
	bHab13	: BOOL := TRUE;
	iMux13K : INT := 2;
	iMux13R : INT; // valor esperado = 30		

// Variáveis para testar LIMIT
	bHab14	: BOOL := TRUE;
	iLim14In : INT := 5;
	iLim14R : INT; // valor esperado = 20		
	
// Variáveis para testar MOVE
	bHab15	: BOOL := TRUE;
	iMov15In : INT := 5;
	iMov15R : INT; // valor esperado = 5
	
// Variáveis para testar Conversão
	bHab16	: BOOL := TRUE;
	iConv16R : INT; // valor esperado = 1	
	
// Variáveis para testar elementos Ladder
	bContato01 : BOOL := TRUE;  
	bContato01R : BOOL;  // valor esperado = 1	
	
	bContato02 : BOOL := FALSE;  
	bContato02R : BOOL;  // valor esperado = 1	

	bContato03 : BOOL := TRUE;  
	bContato03R : BOOL;  // valor esperado = 1	
	
END_VAR

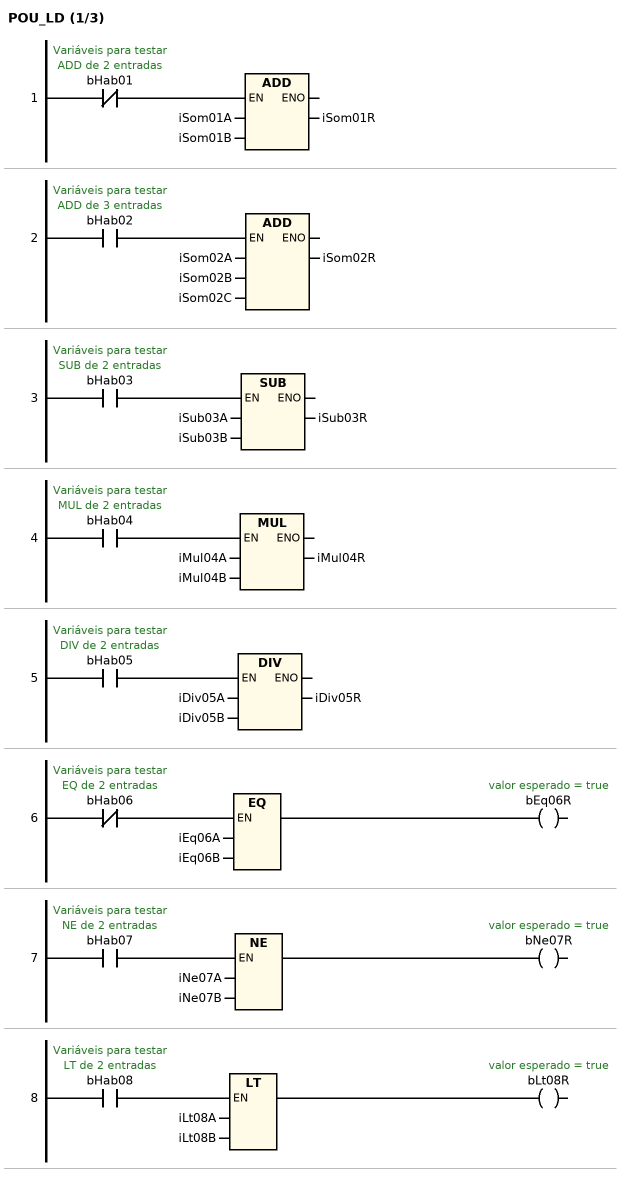
// NETWORK 1
//   bHab01: Variáveis para testar ADD de 2 entradas
IF NOT bHab01 THEN iSom01R := iSom01A + iSom01B; END_IF

// NETWORK 2
//   bHab02: Variáveis para testar ADD de 3 entradas
IF bHab02 THEN iSom02R := iSom02A + iSom02B + iSom02C; END_IF

// NETWORK 3
//   bHab03: Variáveis para testar SUB de 2 entradas
IF bHab03 THEN iSub03R := iSub03A - iSub03B; END_IF

// NETWORK 4
//   bHab04: Variáveis para testar MUL de 2 entradas
IF bHab04 THEN iMul04R := iMul04A * iMul04B; END_IF

// NETWORK 5
//   bHab05: Variáveis para testar DIV de 2 entradas
IF bHab05 THEN iDiv05R := iDiv05A / iDiv05B; END_IF

// NETWORK 6
//   bHab06: Variáveis para testar EQ de 2 entradas
//   bEq06R: valor esperado = true
bEq06R := NOT bHab06 AND iEq06A = iEq06B;

// NETWORK 7
//   bHab07: Variáveis para testar NE de 2 entradas
//   bNe07R: valor esperado = true
bNe07R := bHab07 AND iNe07A <> iNe07B;

// NETWORK 8
//   bHab08: Variáveis para testar LT de 2 entradas
//   bLt08R: valor esperado = true
bLt08R := bHab08 AND iLt08A < iLt08B;

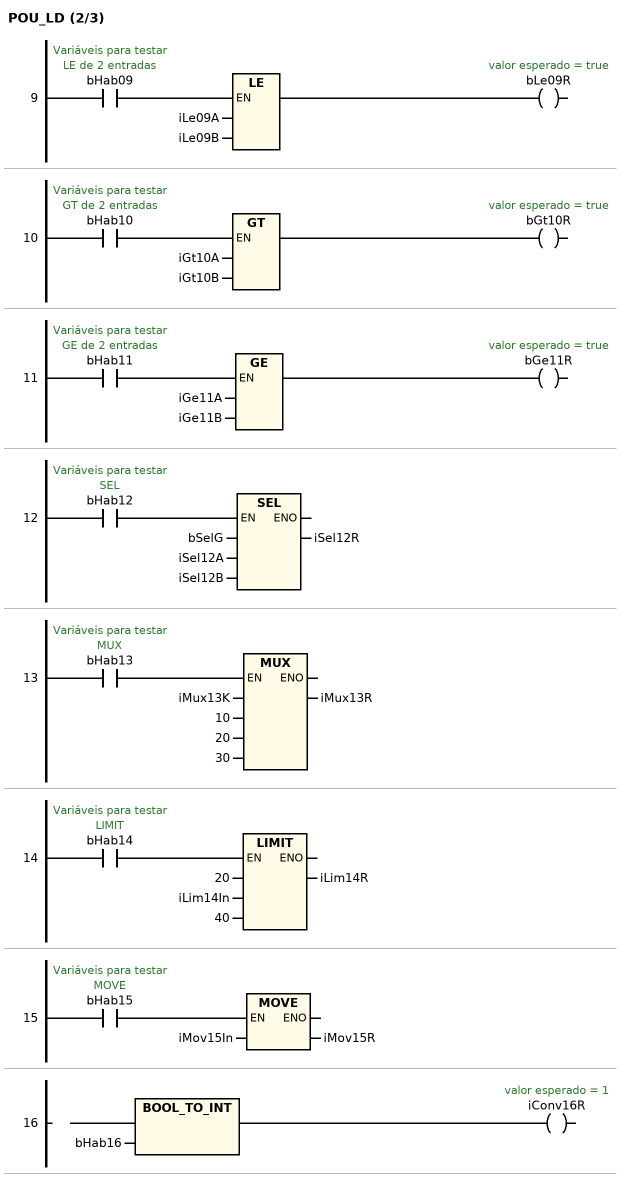
// NETWORK 9
//   bHab09: Variáveis para testar LE de 2 entradas
//   bLe09R: valor esperado = true
bLe09R := bHab09 AND iLe09A <= iLe09B;

// NETWORK 10
//   bHab10: Variáveis para testar GT de 2 entradas
//   bGt10R: valor esperado = true
bGt10R := bHab10 AND iGt10A > iGt10B;

// NETWORK 11
//   bHab11: Variáveis para testar GE de 2 entradas
//   bGe11R: valor esperado = true
bGe11R := bHab11 AND iGe11A >= iGe11B;

// NETWORK 12
//   bHab12: Variáveis para testar SEL
IF bHab12 THEN iSel12R := SEL(bSelG, iSel12A, iSel12B); END_IF

// NETWORK 13
//   bHab13: Variáveis para testar MUX
IF bHab13 THEN iMux13R := MUX(iMux13K, 10, 20, 30); END_IF

// NETWORK 14
//   bHab14: Variáveis para testar LIMIT
IF bHab14 THEN iLim14R := LIMIT(20, iLim14In, 40); END_IF

// NETWORK 15
//   bHab15: Variáveis para testar MOVE
IF bHab15 THEN iMov15R := iMov15In; END_IF

// NETWORK 16
//   bHab16: Variáveis para testar Conversão
//   iConv16R: valor esperado = 1
iConv16R := BOOL_TO_INT(bHab16);

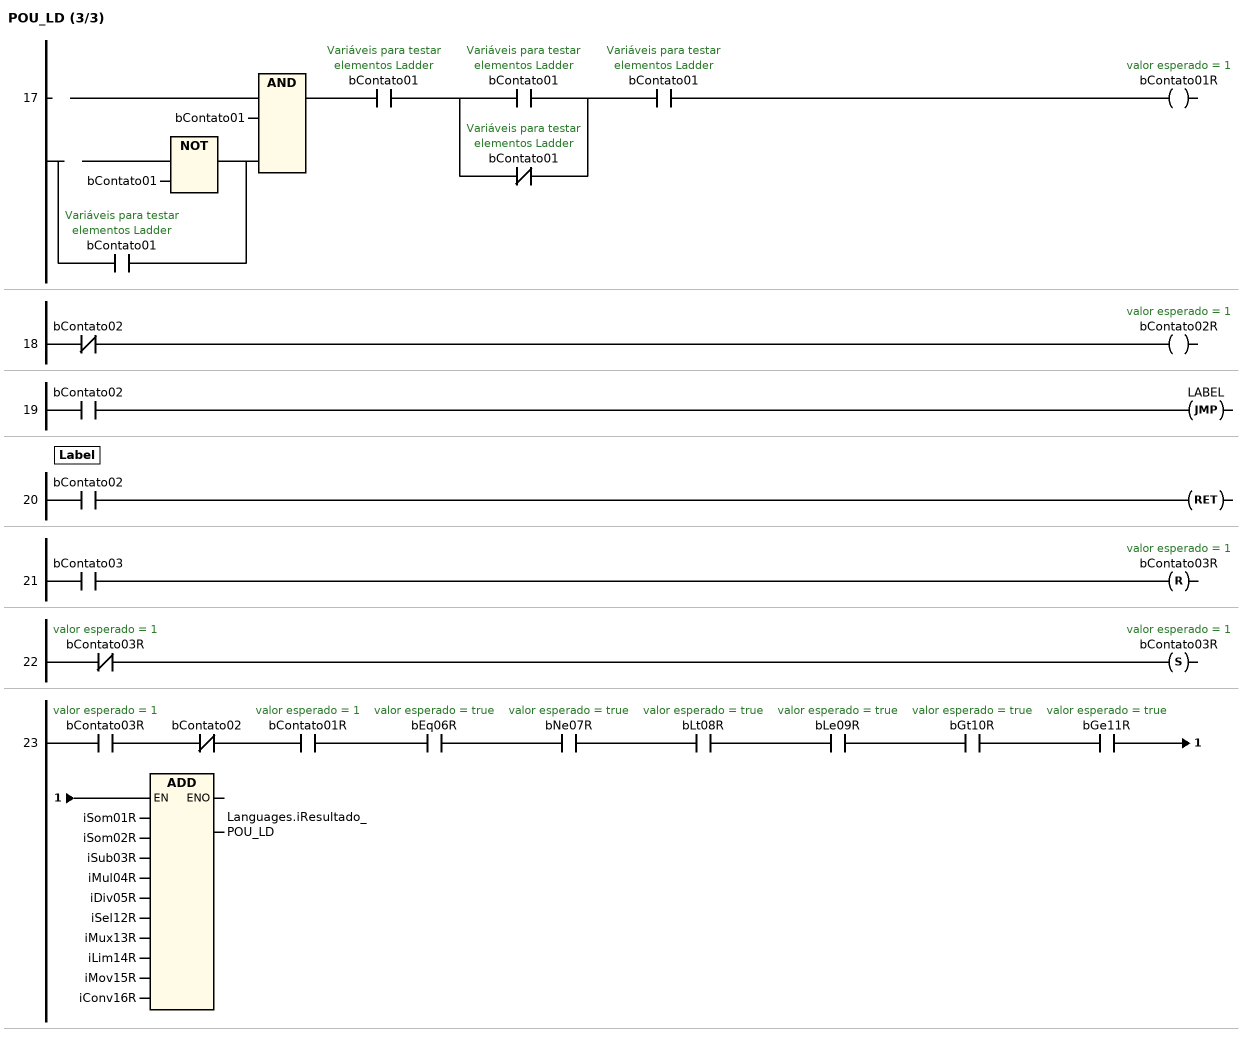
// NETWORK 17
//   bContato01: Variáveis para testar elementos Ladder
//   bContato01R: valor esperado = 1
bContato01R := (((bContato01 AND (NOT bContato01 OR bContato01)) AND bContato01) AND (bContato01 OR NOT bContato01)) AND bContato01;

// NETWORK 18
//   bContato02R: valor esperado = 1
bContato02R := NOT bContato02;

// NETWORK 19
IF bContato02 THEN JMP LABEL; END_IF

// NETWORK 20
Label:
IF bContato02 THEN RETURN; END_IF

// NETWORK 21
//   bContato03R: valor esperado = 1
bContato03R R= bContato03;

// NETWORK 22
//   bContato03R: valor esperado = 1
bContato03R S= NOT bContato03R;

// NETWORK 23
//   bContato03R: valor esperado = 1
//   bContato01R: valor esperado = 1
//   bEq06R: valor esperado = true
//   bNe07R: valor esperado = true
//   bLt08R: valor esperado = true
//   bLe09R: valor esperado = true
//   bGt10R: valor esperado = true
//   bGe11R: valor esperado = true
//   iSom01R: valor esperado = 3
//   iSom02R: valor esperado = 6
//   iSub03R: valor esperado = 1
//   iMul04R: valor esperado = 16
//   iDiv05R: valor esperado = 4
//   iSel12R: valor esperado = 26
//   iMux13R: valor esperado = 30
//   iLim14R: valor esperado = 20
//   iMov15R: valor esperado = 5
//   iConv16R: valor esperado = 1
IF bContato03R AND NOT bContato02 AND bContato01R AND bEq06R AND bNe07R AND bLt08R AND bLe09R AND bGt10R AND bGe11R THEN
    Languages.iResultado_POU_LD := iSom01R + iSom02R + iSub03R + iMul04R + iDiv05R + iSel12R + iMux13R + iLim14R + iMov15R + iConv16R;
END_IF

END_PROGRAM

// Device/Application/UserPOUs/Redundant/Languages/POU_IL
PROGRAM POU_IL
VAR



// Variáveis para testar ADD de 2 entradas
	iSom01A	: INT :=1;
	iSom01B : INT :=2;
	iSom01R : INT; // valor esperado = 3
	
// Variáveis para testar ADD de 3 entradas
	iSom02A	: INT :=1;
	iSom02B : INT :=2;
	iSom02C : INT :=3;
	iSom02R : INT; // valor esperado = 6
	
// Variáveis para testar SUB de 2 entradas
	iSub03A	: INT :=3;
	iSub03B : INT :=2;
	iSub03R : INT; // valor esperado = 1
	
// Variáveis para testar MUL de 2 entradas
	iMul04A	: INT :=4;
	iMul04B : INT :=4;
	iMul04R : INT; // valor esperado = 16
	
// Variáveis para testar DIV de 2 entradas
	iDiv05A	: INT :=20;
	iDiv05B : INT :=5;
	iDiv05R : INT; // valor esperado = 4
	
// Variáveis para testar EQ de 2 entradas
	iEq06A	: INT :=25;
	iEq06B : INT :=25;
	bEq06R : BOOL; // valor esperado = true	
	iEq06R : INT; // valor esperado = 1

// Variáveis para testar NE de 2 entradas
	iNe07A	: INT :=24;
	iNe07B : INT :=25;
	bNe07R : BOOL; // valor esperado = true
	iNe07R : INT; // valor esperado = 1

// Variáveis para testar LT de 2 entradas
	iLt08A	: INT :=24;
	iLt08B : INT :=25;
	bLt08R : BOOL; // valor esperado = true		
	iLt08R : INT; // valor esperado = 1		
	
// Variáveis para testar LE de 2 entradas
	iLe09A	: INT :=25;
	iLe09B : INT :=25;
	bLe09R : BOOL; // valor esperado = true		
	iLe09R : INT; // valor esperado = 1
	
// Variáveis para testar GT de 2 entradas
	iGt10A	: INT :=26;
	iGt10B : INT :=25;
	bGt10R : BOOL; // valor esperado = true	
	iGt10R : INT; // valor esperado = 1	

// Variáveis para testar GE de 2 entradas
	iGe11A	: INT :=26;
	iGe11B : INT :=26;
	bGe11R : BOOL; // valor esperado = true		
	iGe11R : INT; // valor esperado = 1	
	
// Variáveis para testar SEL
	bSelG : BOOL := TRUE;
	iSel12A	: INT :=20;
	iSel12B : INT :=26;
	iSel12R : INT; // valor esperado = 26		
	
// Variáveis para testar MUX
	iMux13K : INT := 2;
	iMux13R : INT; // valor esperado = 30		

// Variáveis para testar LIMIT
	iLim14In : INT := 5;
	iLim14R : INT; // valor esperado = 20		
	
// Variáveis para testar MOVE
	iMov15In : INT := 5;
	iMov15R : INT; // valor esperado = 5
	
// Variáveis para testar Conversão
	bHab16	: BOOL := TRUE;
	iConv16R : INT; // valor esperado = 1	
	
// Variáveis para testar elementos Ladder
	bContato01 : BOOL := TRUE;  
	bContato01R : BOOL;  // valor esperado = 1	
	
	bContato02 : BOOL := FALSE;  
	bContato02R : BOOL;  // valor esperado = 1	

	bContato03 : BOOL := TRUE;  
	bContato03R : BOOL;  // valor esperado = 1	
	
END_VAR

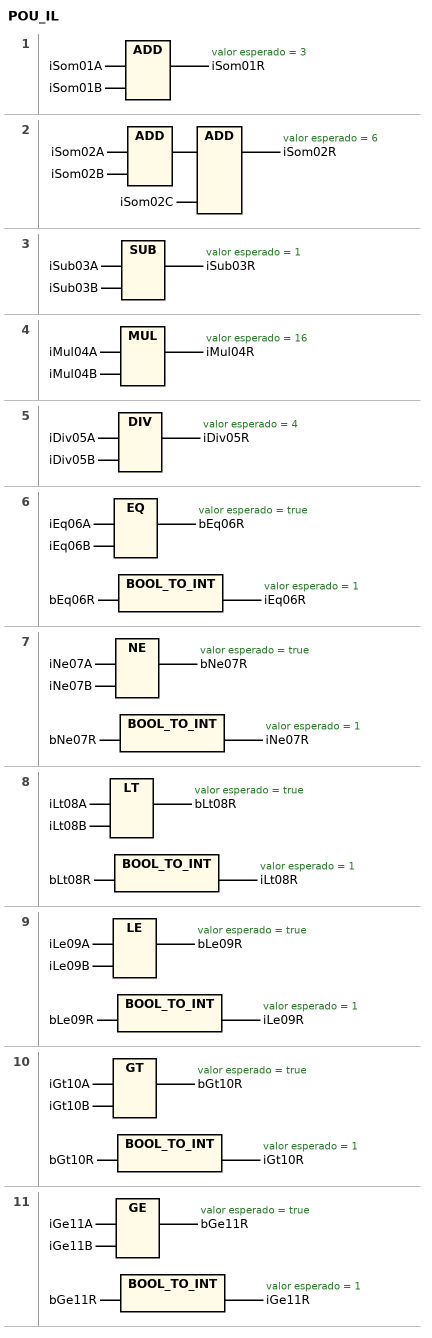
// NETWORK 1
//   iSom01R: valor esperado = 3
iSom01R := iSom01A + iSom01B;

// NETWORK 2
//   iSom02R: valor esperado = 6
iSom02R := (iSom02A + iSom02B) + iSom02C;

// NETWORK 3
//   iSub03R: valor esperado = 1
iSub03R := iSub03A - iSub03B;

// NETWORK 4
//   iMul04R: valor esperado = 16
iMul04R := iMul04A * iMul04B;

// NETWORK 5
//   iDiv05R: valor esperado = 4
iDiv05R := iDiv05A / iDiv05B;

// NETWORK 6
//   bEq06R: valor esperado = true
//   iEq06R: valor esperado = 1
bEq06R := iEq06A = iEq06B;
iEq06R := BOOL_TO_INT(bEq06R);

// NETWORK 7
//   bNe07R: valor esperado = true
//   iNe07R: valor esperado = 1
bNe07R := iNe07A <> iNe07B;
iNe07R := BOOL_TO_INT(bNe07R);

// NETWORK 8
//   bLt08R: valor esperado = true
//   iLt08R: valor esperado = 1
bLt08R := iLt08A < iLt08B;
iLt08R := BOOL_TO_INT(bLt08R);

// NETWORK 9
//   bLe09R: valor esperado = true
//   iLe09R: valor esperado = 1
bLe09R := iLe09A <= iLe09B;
iLe09R := BOOL_TO_INT(bLe09R);

// NETWORK 10
//   bGt10R: valor esperado = true
//   iGt10R: valor esperado = 1
bGt10R := iGt10A > iGt10B;
iGt10R := BOOL_TO_INT(bGt10R);

// NETWORK 11
//   bGe11R: valor esperado = true
//   iGe11R: valor esperado = 1
bGe11R := iGe11A >= iGe11B;
iGe11R := BOOL_TO_INT(bGe11R);

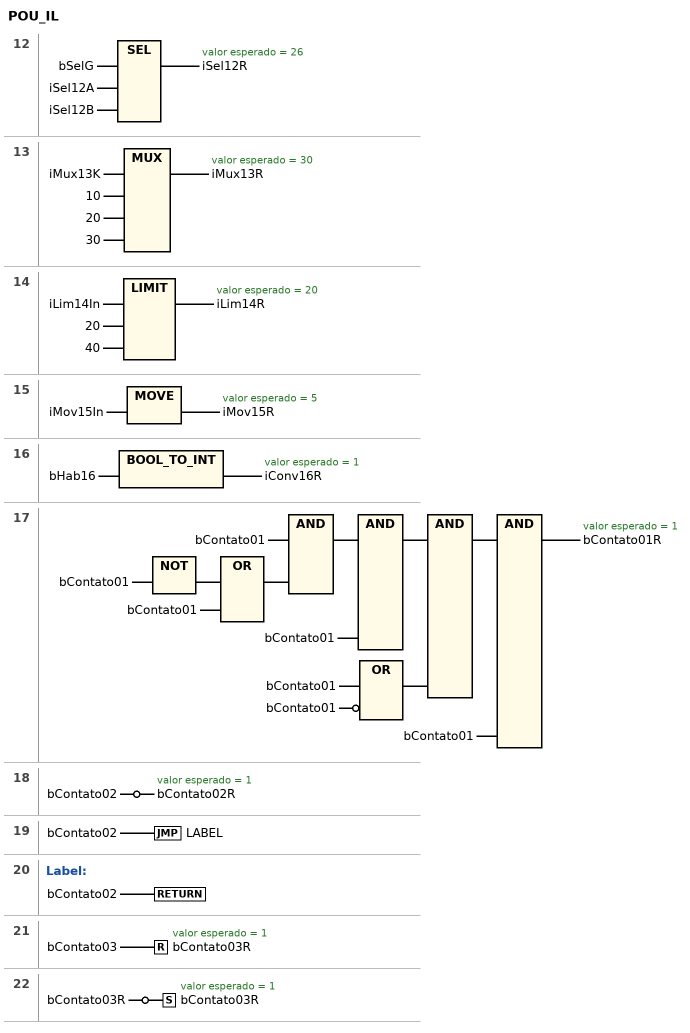
// NETWORK 12
//   iSel12R: valor esperado = 26
iSel12R := SEL(bSelG, iSel12A, iSel12B);

// NETWORK 13
//   iMux13R: valor esperado = 30
iMux13R := MUX(iMux13K, 10, 20, 30);

// NETWORK 14
//   iLim14R: valor esperado = 20
iLim14R := LIMIT(iLim14In, 20, 40);

// NETWORK 15
//   iMov15R: valor esperado = 5
iMov15R := iMov15In;

// NETWORK 16
//   iConv16R: valor esperado = 1
iConv16R := BOOL_TO_INT(bHab16);

// NETWORK 17
//   bContato01R: valor esperado = 1
bContato01R := (((bContato01 AND (NOT bContato01 OR bContato01)) AND bContato01) AND (bContato01 OR NOT bContato01)) AND bContato01;

// NETWORK 18
//   bContato02R: valor esperado = 1
bContato02R := NOT bContato02;

// NETWORK 19
IF bContato02 THEN JMP LABEL; END_IF

// NETWORK 20
Label:
IF bContato02 THEN RETURN; END_IF

// NETWORK 21
//   bContato03R: valor esperado = 1
bContato03R R= bContato03;

// NETWORK 22
//   bContato03R: valor esperado = 1
bContato03R S= NOT bContato03R;

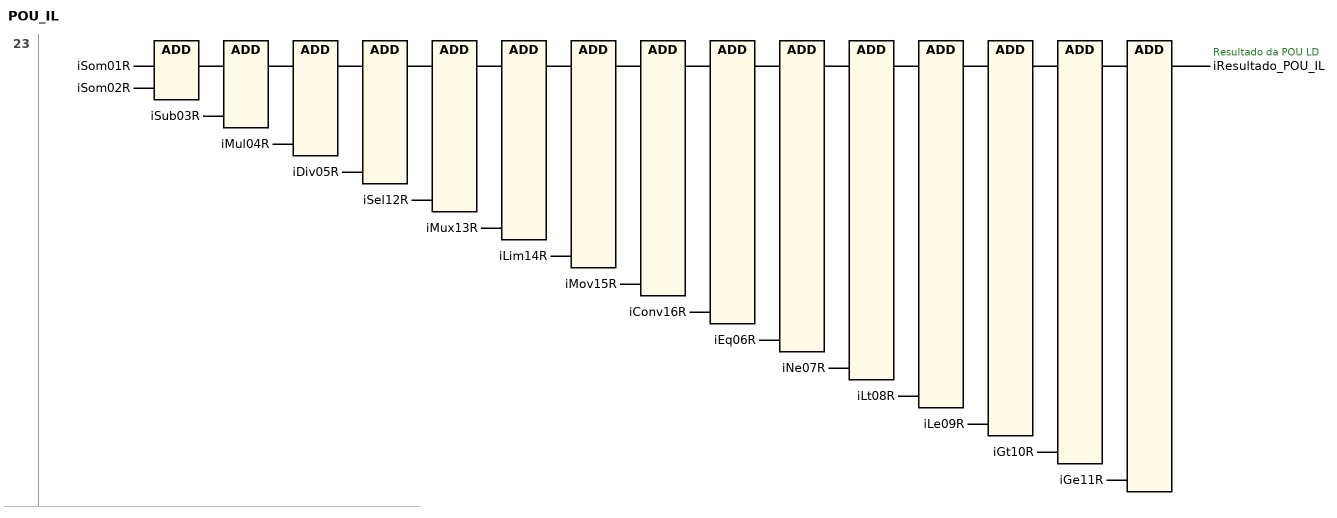
// NETWORK 23
//   iResultado_POU_IL: Resultado da POU LD
iResultado_POU_IL := ((((((((((((((iSom01R + iSom02R) + iSub03R) + iMul04R) + iDiv05R) + iSel12R) + iMux13R) + iLim14R) + iMov15R) + iConv16R) + iEq06R) + iNe07R) + iLt08R) + iLe09R) + iGt10R) + iGe11R;

END_PROGRAM

// Device/Application/UserPOUs/Redundant/Languages/POU_CFC
PROGRAM POU_CFC
VAR
	/// Variáveis para testar ADD de 2 entradas
	bHab01: BOOL := FALSE;
	iSom01A: INT := 1;
	iSom01B: INT := 2;
	/// valor esperado = 3
	iSom01R: INT;
	/// Variáveis para testar SUB de 2 entradas
	bHab03: BOOL := TRUE;
	iSub03A: INT := 3;
	iSub03B: INT := 2;
	/// valor esperado = 1
	iSub03R: INT;
	/// Variáveis para testar MUL de 2 entradas
	bHab04: BOOL := TRUE;
	iMul04A: INT := 4;
	iMul04B: INT := 4;
	/// valor esperado = 16
	iMul04R: INT;
	/// Variáveis para testar DIV de 2 entradas
	bHab05: BOOL := TRUE;
	iDiv05A: INT := 20;
	iDiv05B: INT := 5;
	/// valor esperado = 4
	iDiv05R: INT;
	/// Variáveis para testar EQ de 2 entradas
	bHab06: BOOL := FALSE;
	iEq06A: INT := 25;
	iEq06B: INT := 25;
	/// valor esperado = true	
	bEq06R: BOOL;
	/// valor esperado= 1
	iEq06R: INT;
	/// Variáveis para testar NE de 2 entradas
	bHab07: BOOL := TRUE;
	iNe07A: INT := 24;
	iNe07B: INT := 25;
	/// valor esperado = true
	bNe07R: BOOL;
	/// valor esperado= 1
	iNe07R: INT;
	/// Variáveis para testar LT de 2 entradas
	bHab08: BOOL := TRUE;
	iLt08A: INT := 24;
	iLt08B: INT := 25;
	/// valor esperado = true		
	bLt08R: BOOL;
	/// valor esperado= 1		
	iLt08R: INT;
	/// Variáveis para testar LE de 2 entradas
	bHab09: BOOL := TRUE;
	iLe09A: INT := 25;
	iLe09B: INT := 25;
	/// valor esperado = true		
	bLe09R: BOOL;
	/// valor esperado= 1			
	iLe09R: INT;
	/// Variáveis para testar GT de 2 entradas
	bHab10: BOOL := TRUE;
	iGt10A: INT := 26;
	iGt10B: INT := 25;
	/// valor esperado = true	
	bGt10R: BOOL;
	/// valor esperado= 1
	iGt10R: INT;
	/// Variáveis para testar GE de 2 entradas
	bHab11: BOOL := TRUE;
	iGe11A: INT := 26;
	iGe11B: INT := 26;
	/// valor esperado = true		
	bGe11R: BOOL;
	/// valor esperado= 1
	iGe11R: INT;
	/// Variáveis para testar SEL
	bHab12: BOOL := TRUE;
	bSelG: BOOL := TRUE;
	iSel12A: INT := 20;
	iSel12B: INT := 26;
	/// valor esperado = 26		
	iSel12R: INT;
	/// Variáveis para testar MUX
	bHab13: BOOL := FALSE;
	iMux13K: INT := 2;
	/// valor esperado = 30		
	iMux13R: INT;
	/// Variáveis para testar LIMIT
	bHab14: BOOL := TRUE;
	iLim14In: INT := 5;
	/// valor esperado = 20		
	iLim14R: INT;
	/// Variáveis para testar MOVE
	bHab15: BOOL := TRUE;
	iMov15In: INT := 5;
	/// valor esperado = 5
	iMov15R: INT;
	/// Variáveis para testar Conversão
	bHab16: BOOL := TRUE;
	/// valor esperado = 1	
	iConv16R: INT;
	/// Variáveis para testar Composer
	iComp_InA: INT := 10;
	iComp_InB: INT := 33;
	fb_FB_CFC: FB_CFC;
	/// valor esperado 11
	iComp_OutA: INT;
	/// valor esperado 35	
	iComp_OutB: INT;
	/// Variáveis para testar Seletor
	iSele_InA: INT := 5;
	fb_FB_CFC_02: FB_CFC_2;
	/// valor esperado 15
	iSele_OutA: INT;
	/// valor esperado 25	
	iSele_OutB: INT;
	// Chamada de function block para fazer teste de reordenação online change - Demanda: 23194
	TesteFb:fbTotalizador;
	TesteFbVarInput1:ULINT;
	TesteFbVarInput2:ULINT;

END_VAR
VAR // added by the converter: edge detectors and wires of the graphical bodies
    _s1 : DUT_CFC;
    _w1, _w2, _w3, _w10, _w13, _w14 : INT;
    _w4, _w5, _w6, _w7, _w8, _w9 : BOOL;
    _w11, _w12 : ANY;
END_VAR

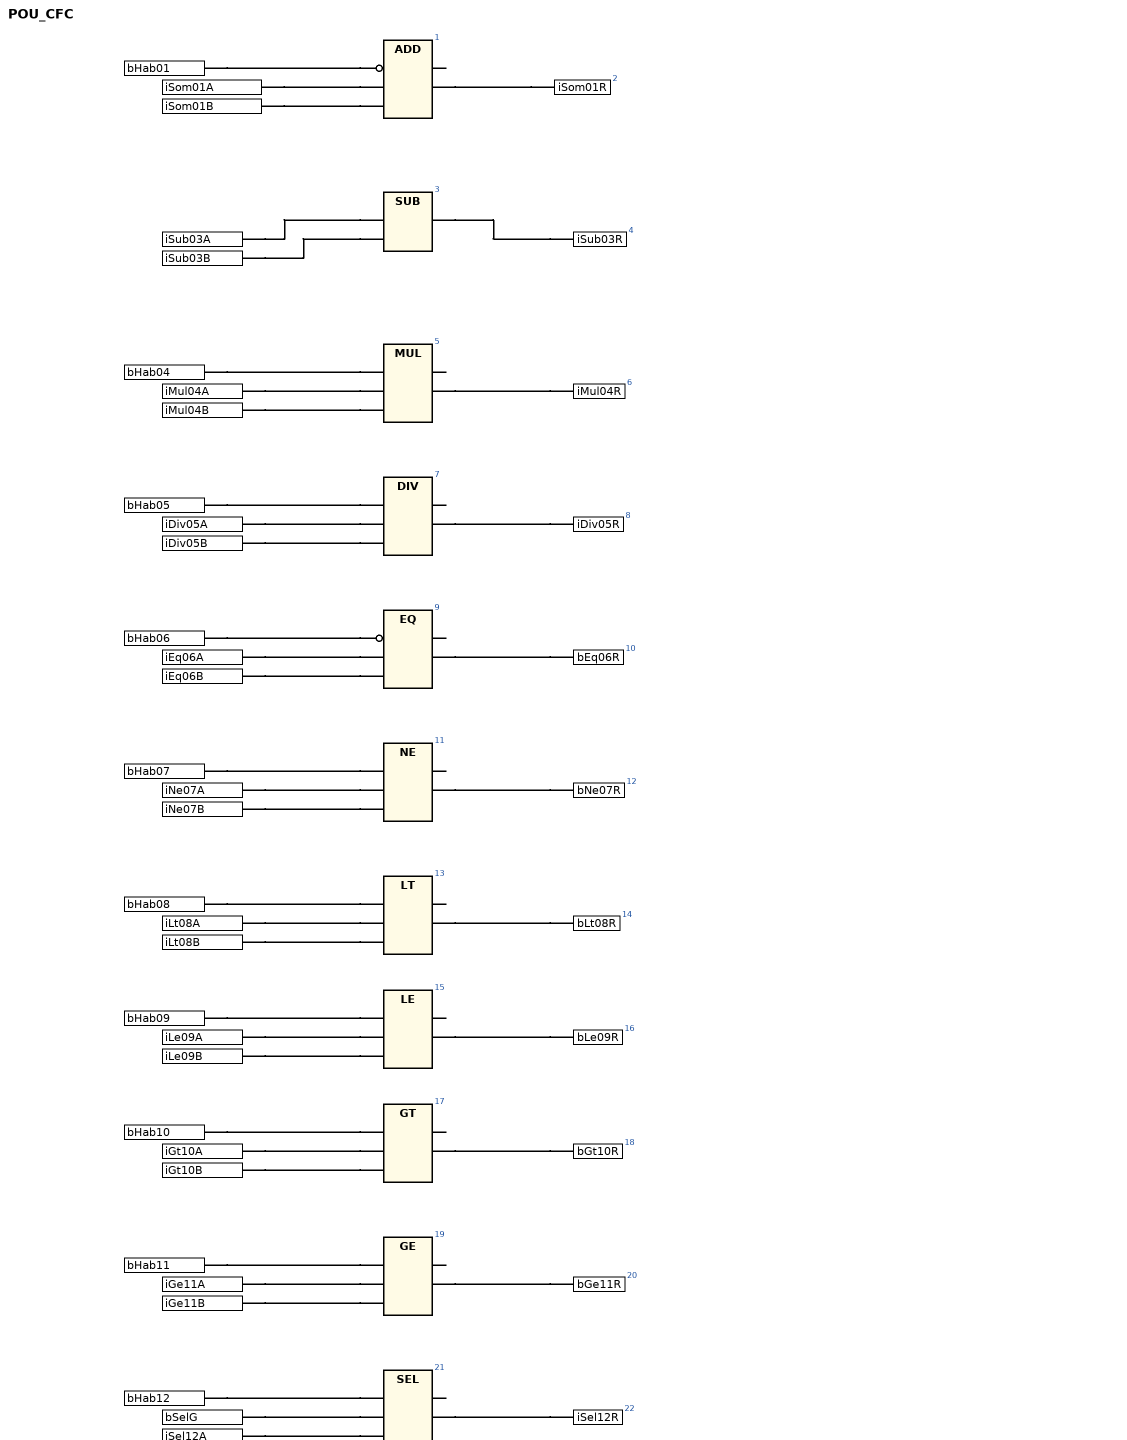
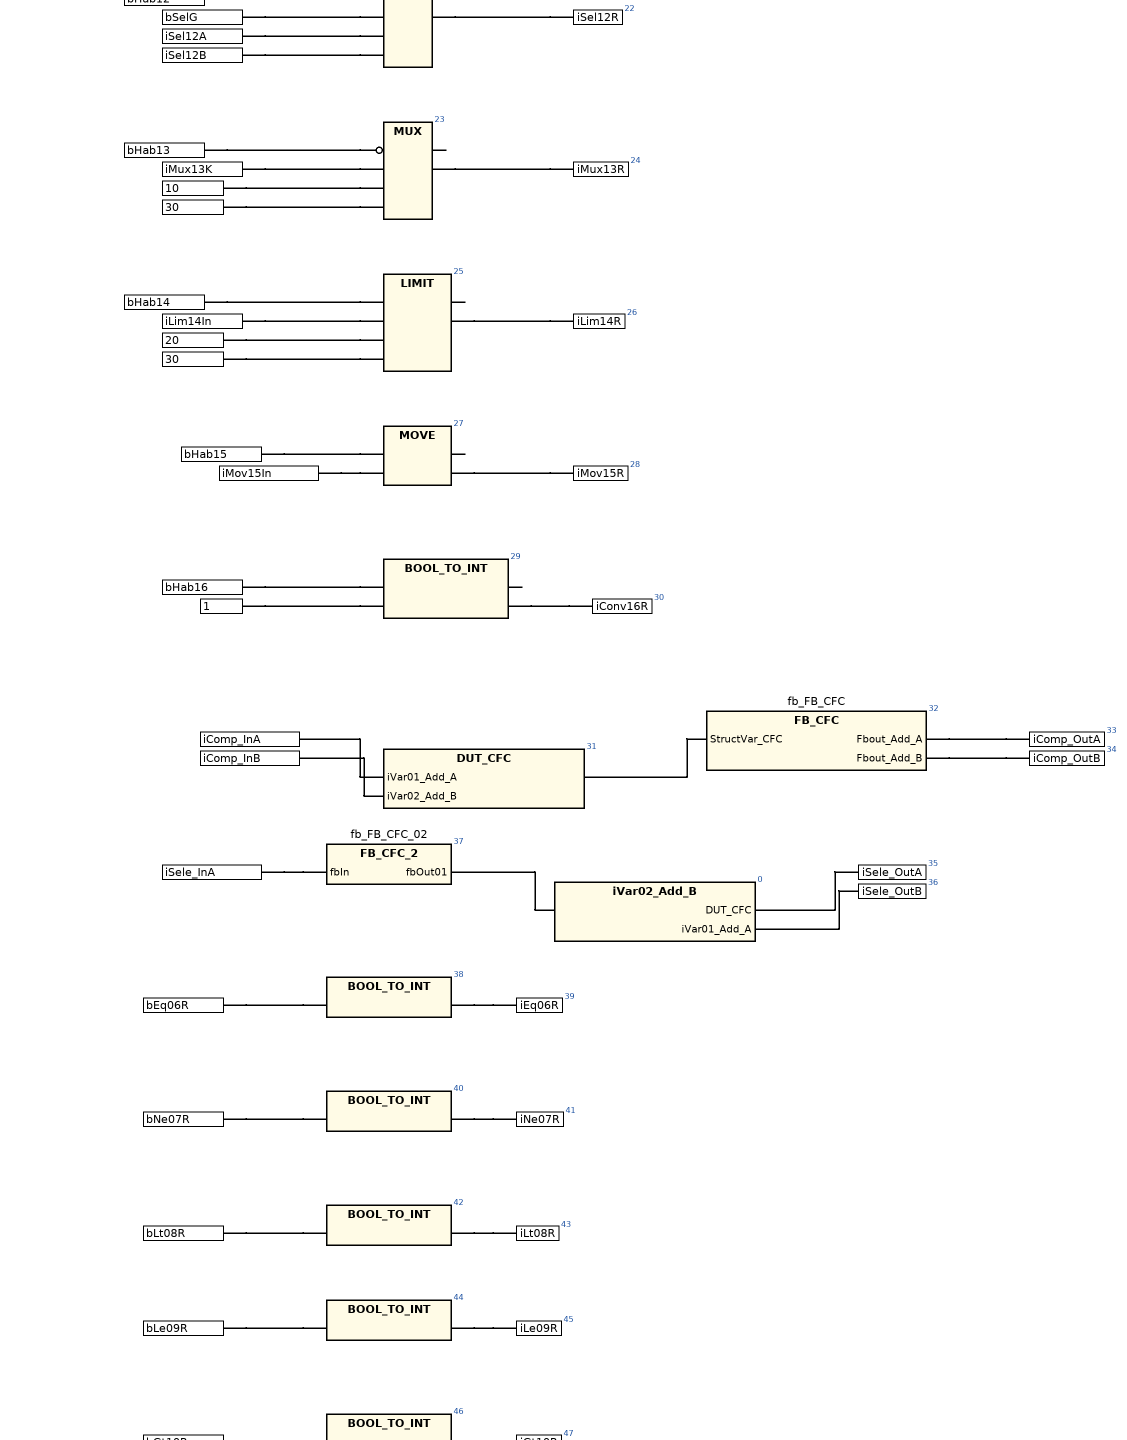
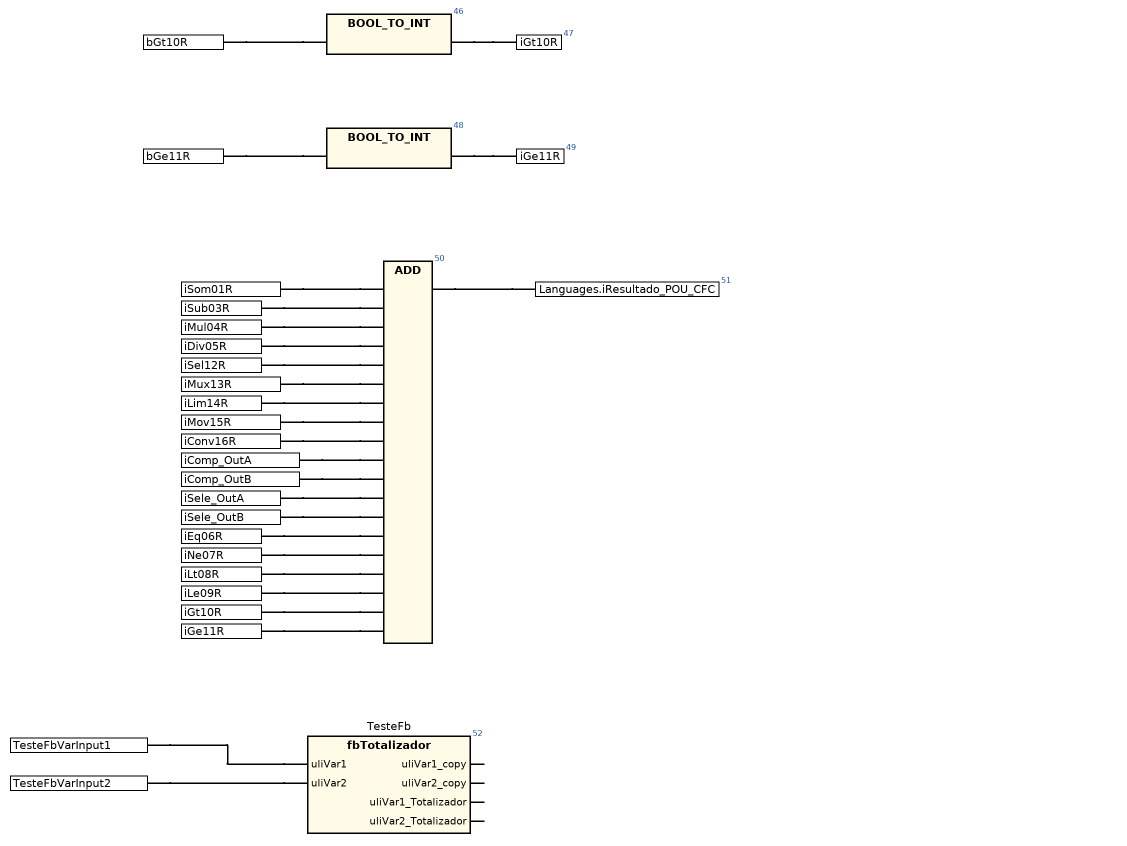
IF NOT bHab01 THEN _w1 := iSom01A + iSom01B; END_IF
iSom01R := _w1;
iSub03R := iSub03A - iSub03B;
IF bHab04 THEN _w2 := iMul04A * iMul04B; END_IF
iMul04R := _w2;
IF bHab05 THEN _w3 := iDiv05A / iDiv05B; END_IF
iDiv05R := _w3;
IF NOT bHab06 THEN _w4 := iEq06A = iEq06B; END_IF
bEq06R := _w4;
IF bHab07 THEN _w5 := iNe07A <> iNe07B; END_IF
bNe07R := _w5;
IF bHab08 THEN _w6 := iLt08A < iLt08B; END_IF
bLt08R := _w6;
IF bHab09 THEN _w7 := iLe09A <= iLe09B; END_IF
bLe09R := _w7;
IF bHab10 THEN _w8 := iGt10A > iGt10B; END_IF
bGt10R := _w8;
IF bHab11 THEN _w9 := iGe11A >= iGe11B; END_IF
bGe11R := _w9;
IF bHab12 THEN _w10 := SEL(bSelG, iSel12A, iSel12B); END_IF
iSel12R := _w10;
IF NOT bHab13 THEN _w11 := MUX(iMux13K, 10, 30); END_IF
iMux13R := _w11;
IF bHab14 THEN _w12 := LIMIT(iLim14In, 20, 30); END_IF
iLim14R := _w12;
IF bHab15 THEN _w13 := iMov15In; END_IF
iMov15R := _w13;
IF bHab16 THEN _w14 := BOOL_TO_INT(1); END_IF
iConv16R := _w14;
// compose _s1 : DUT_CFC
_s1.iVar01_Add_A := iComp_InA;
_s1.iVar02_Add_B := iComp_InB;
fb_FB_CFC(StructVar_CFC := _s1); // FB_CFC
iComp_OutA := fb_FB_CFC.Fbout_Add_A;
iComp_OutB := fb_FB_CFC.Fbout_Add_B;
iSele_OutA := fb_FB_CFC_02.fbOut01.DUT_CFC;
iSele_OutB := fb_FB_CFC_02.fbOut01.iVar01_Add_A;
fb_FB_CFC_02(fbIn := iSele_InA); // FB_CFC_2
iEq06R := BOOL_TO_INT(bEq06R);
iNe07R := BOOL_TO_INT(bNe07R);
iLt08R := BOOL_TO_INT(bLt08R);
iLe09R := BOOL_TO_INT(bLe09R);
iGt10R := BOOL_TO_INT(bGt10R);
iGe11R := BOOL_TO_INT(bGe11R);
Languages.iResultado_POU_CFC := iSom01R + iSub03R + iMul04R + iDiv05R + iSel12R + iMux13R + iLim14R + iMov15R + iConv16R + iComp_OutA + iComp_OutB + iSele_OutA + iSele_OutB + iEq06R + iNe07R + iLt08R + iLe09R + iGt10R + iGe11R;
TesteFb(uliVar1 := TesteFbVarInput1, uliVar2 := TesteFbVarInput2); // fbTotalizador

END_PROGRAM

// Device/Application/UserPOUs/Redundant/Languages/CFC/FB_CFC
FUNCTION_BLOCK FB_CFC
VAR_INPUT
	StructVar_CFC: DUT_CFC;
END_VAR
VAR_OUTPUT
	Fbout_Add_A: INT;
	Fbout_Add_B: INT;
END_VAR

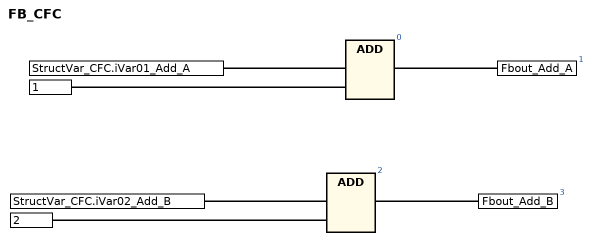
Fbout_Add_A := StructVar_CFC.iVar01_Add_A + 1;
Fbout_Add_B := StructVar_CFC.iVar02_Add_B + 2;

END_FUNCTION_BLOCK

// Device/Application/UserPOUs/Redundant/Languages/CFC/FB_CFC_2
FUNCTION_BLOCK FB_CFC_2
VAR_INPUT
	fbIn: INT;
END_VAR
VAR_OUTPUT
	fbOut01: DUT_CFC;
END_VAR

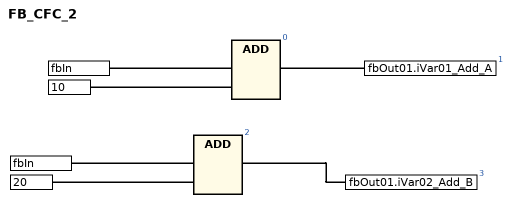
fbOut01.iVar01_Add_A := fbIn + 10;
fbOut01.iVar02_Add_B := fbIn + 20;

END_FUNCTION_BLOCK

// Device/Application/UserFunctionsBlocks/fbTotalizador
FUNCTION_BLOCK fbTotalizador
VAR_INPUT
	
	uliVar1: ULINT;
	uliVar2: ULINT;
	
END_VAR
VAR_OUTPUT
	
	uliVar1_copy: ULINT;
	uliVar2_copy:ULINT;
	uliVar1_Totalizador:ULINT;
	uliVar2_Totalizador:ULINT;
END_VAR
VAR
END_VAR

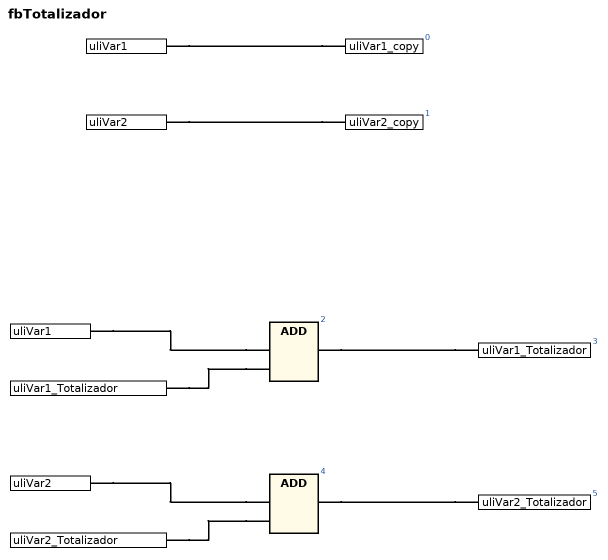
uliVar1_copy := uliVar1;
uliVar2_copy := uliVar2;
uliVar1_Totalizador := uliVar1 + uliVar1_Totalizador;
uliVar2_Totalizador := uliVar2 + uliVar2_Totalizador;

END_FUNCTION_BLOCK

// Device/Application/UserPOUs/Redundant/Languages/CFC/POU_CFC_1000
PROGRAM POU_CFC_1000
//Esta POU existe para tetar lógica com mais de 1000 sequencias, poi so projeto da Petrobras usam em torno de 800 sequencias e já apresentou problemas com isso.
VAR
	iInt: INT;
END_VAR
VAR // added by the converter: edge detectors and wires of the graphical bodies
    _w1, _w2, _w3, _w4, _w5, _w6, _w7, _w8, _w9, _w10, _w11, _w12, _w13, _w14, _w15, _w16, _w17, _w18, _w19, _w20, _w21, _w22, _w23, _w24, _w25, _w26, _w27, _w28, _w29, _w30, _w31, _w32, _w33, _w34, _w35, _w36, _w37, _w38, _w39, _w40, _w41, _w42, _w43, _w44, _w45, _w46, _w47, _w48, _w49, _w50, _w51, _w52, _w53, _w54, _w55, _w56, _w57, _w58, _w59, _w60, _w61, _w62, _w63, _w64, _w65, _w66, _w67, _w68, _w69, _w70, _w71, _w72, _w73, _w74, _w75, _w76, _w77, _w78, _w79, _w80, _w81, _w82, _w83, _w84, _w85, _w86, _w87, _w88, _w89, _w90, _w91, _w92, _w93, _w94, _w95, _w96, _w97, _w98, _w99, _w100, _w101, _w102, _w103, _w104, _w105, _w106, _w107, _w108, _w109, _w110, _w111, _w112, _w113, _w114, _w115, _w116, _w117, _w118, _w119, _w120, _w121, _w122, _w123, _w124, _w125, _w126, _w127, _w128, _w129, _w130, _w131, _w132, _w133, _w134, _w135, _w136, _w137, _w138, _w139, _w140, _w141, _w142, _w143, _w144, _w145, _w146, _w147, _w148, _w149, _w150, _w151, _w152, _w153, _w154, _w155, _w156, _w157, _w158, _w159, _w160, _w161, _w162, _w163, _w164, _w165, _w166, _w167, _w168, _w169, _w170, _w171, _w172, _w173, _w174, _w175, _w176, _w177, _w178, _w179, _w180, _w181, _w182, _w183, _w184, _w185, _w186, _w187, _w188, _w189, _w190, _w191, _w192, _w193, _w194, _w195, _w196, _w197, _w198, _w199, _w200, _w201, _w202, _w203, _w204, _w205, _w206, _w207, _w208, _w209, _w210, _w211, _w212, _w213, _w214, _w215, _w216, _w217, _w218, _w219, _w220, _w221, _w222, _w223, _w224, _w225, _w226, _w227, _w228, _w229, _w230, _w231, _w232, _w233, _w234, _w235, _w236, _w237, _w238, _w239, _w240, _w241, _w242, _w243, _w244, _w245, _w246, _w247, _w248, _w249, _w250, _w251, _w252, _w253, _w254, _w255, _w256, _w257, _w258, _w259, _w260, _w261, _w262, _w263, _w264, _w265, _w266, _w267, _w268, _w269, _w270, _w271, _w272, _w273, _w274, _w275, _w276, _w277, _w278, _w279, _w280, _w281, _w282, _w283, _w284, _w285, _w286, _w287, _w288, _w289, _w290, _w291, _w292, _w293, _w294, _w295, _w296, _w297, _w298, _w299, _w300, _w301, _w302, _w303, _w304, _w305, _w306, _w307, _w308, _w309, _w310, _w311, _w312, _w313, _w314, _w315, _w316, _w317, _w318, _w319, _w320, _w321, _w322, _w323, _w324, _w325, _w326, _w327, _w328, _w329, _w330, _w331, _w332, _w333, _w334, _w335, _w336, _w337, _w338, _w339, _w340, _w341, _w342, _w343, _w344, _w345, _w346, _w347, _w348, _w349, _w350, _w351, _w352, _w353, _w354, _w355, _w356, _w357, _w358, _w359, _w360, _w361, _w362, _w363, _w364, _w365, _w366, _w367, _w368, _w369, _w370, _w371, _w372, _w373, _w374, _w375, _w376, _w377, _w378, _w379, _w380, _w381, _w382, _w383, _w384, _w385, _w386, _w387, _w388, _w389, _w390, _w391, _w392, _w393, _w394, _w395, _w396, _w397, _w398, _w399, _w400, _w401, _w402, _w403, _w404, _w405, _w406, _w407, _w408, _w409, _w410, _w411, _w412, _w413, _w414, _w415, _w416, _w417, _w418, _w419, _w420, _w421, _w422, _w423, _w424, _w425, _w426, _w427, _w428, _w429, _w430, _w431, _w432, _w433, _w434, _w435, _w436, _w437, _w438, _w439, _w440, _w441, _w442, _w443, _w444, _w445, _w446, _w447, _w448, _w449, _w450, _w451, _w452, _w453, _w454, _w455, _w456, _w457, _w458, _w459, _w460, _w461, _w462, _w463, _w464, _w465, _w466, _w467, _w468, _w469, _w470, _w471, _w472, _w473, _w474, _w475, _w476, _w477, _w478, _w479, _w480, _w481, _w482, _w483, _w484, _w485, _w486, _w487, _w488, _w489, _w490, _w491, _w492, _w493, _w494, _w495, _w496, _w497, _w498, _w499, _w500, _w501, _w502, _w503, _w504, _w505, _w506, _w507, _w508, _w509, _w510, _w511, _w512, _w513, _w514, _w515, _w516, _w517, _w518, _w519, _w520, _w521, _w522, _w523, _w524, _w525, _w526, _w527, _w528, _w529, _w530, _w531, _w532, _w533, _w534, _w535, _w536, _w537, _w538, _w539, _w540, _w541, _w542, _w543, _w544, _w545, _w546, _w547, _w548, _w549, _w550, _w551, _w552, _w553, _w554, _w555, _w556, _w557, _w558, _w559, _w560, _w561, _w562, _w563, _w564, _w565, _w566, _w567, _w568, _w569, _w570, _w571, _w572, _w573, _w574, _w575, _w576, _w577, _w578, _w579, _w580, _w581, _w582, _w583, _w584, _w585, _w586, _w587, _w588, _w589, _w590, _w591, _w592, _w593, _w594, _w595, _w596, _w597, _w598, _w599, _w600, _w601, _w602, _w603, _w604, _w605, _w606, _w607, _w608, _w609, _w610, _w611, _w612, _w613, _w614, _w615, _w616, _w617, _w618, _w619, _w620, _w621, _w622, _w623, _w624, _w625, _w626, _w627, _w628, _w629, _w630, _w631, _w632, _w633, _w634, _w635, _w636, _w637, _w638, _w639, _w640, _w641, _w642, _w643, _w644, _w645, _w646, _w647, _w648, _w649, _w650, _w651, _w652, _w653, _w654, _w655, _w656, _w657, _w658, _w659, _w660, _w661, _w662, _w663, _w664, _w665, _w666, _w667, _w668, _w669, _w670, _w671, _w672, _w673, _w674, _w675, _w676, _w677, _w678, _w679, _w680, _w681, _w682, _w683, _w684, _w685, _w686, _w687, _w688, _w689, _w690, _w691, _w692, _w693, _w694, _w695, _w696, _w697, _w698, _w699, _w700, _w701, _w702, _w703, _w704, _w705, _w706, _w707, _w708, _w709, _w710, _w711, _w712, _w713, _w714, _w715, _w716, _w717, _w718, _w719, _w720, _w721, _w722, _w723, _w724, _w725, _w726, _w727, _w728, _w729, _w730, _w731, _w732, _w733, _w734, _w735, _w736, _w737, _w738, _w739, _w740, _w741, _w742, _w743, _w744, _w745, _w746, _w747, _w748, _w749, _w750, _w751, _w752, _w753, _w754, _w755, _w756, _w757, _w758, _w759, _w760, _w761, _w762, _w763, _w764, _w765, _w766, _w767, _w768, _w769, _w770, _w771, _w772, _w773, _w774, _w775, _w776, _w777, _w778, _w779, _w780, _w781, _w782, _w783, _w784, _w785, _w786, _w787, _w788, _w789, _w790, _w791, _w792, _w793, _w794, _w795, _w796, _w797, _w798, _w799, _w800, _w801, _w802, _w803, _w804, _w805, _w806, _w807, _w808, _w809, _w810, _w811, _w812, _w813, _w814, _w815, _w816, _w817, _w818, _w819, _w820, _w821, _w822, _w823, _w824, _w825, _w826, _w827, _w828, _w829, _w830, _w831, _w832, _w833, _w834, _w835, _w836, _w837, _w838, _w839, _w840, _w841, _w842, _w843, _w844, _w845, _w846, _w847, _w848, _w849, _w850, _w851, _w852, _w853, _w854, _w855, _w856, _w857, _w858, _w859, _w860, _w861, _w862, _w863, _w864, _w865, _w866, _w867, _w868, _w869, _w870, _w871, _w872, _w873, _w874, _w875, _w876, _w877, _w878, _w879, _w880, _w881, _w882, _w883, _w884, _w885, _w886, _w887, _w888, _w889, _w890, _w891, _w892, _w893, _w894, _w895, _w896, _w897, _w898, _w899, _w900, _w901, _w902, _w903, _w904, _w905, _w906, _w907, _w908, _w909, _w910, _w911, _w912, _w913, _w914, _w915, _w916, _w917, _w918, _w919, _w920, _w921, _w922, _w923, _w924, _w925, _w926, _w927, _w928, _w929, _w930, _w931, _w932, _w933, _w934, _w935, _w936, _w937, _w938, _w939, _w940, _w941, _w942, _w943, _w944, _w945, _w946, _w947, _w948, _w949, _w950, _w951, _w952, _w953, _w954, _w955, _w956, _w957, _w958, _w959, _w960, _w961, _w962, _w963, _w964, _w965, _w966, _w967, _w968, _w969, _w970, _w971, _w972, _w973, _w974, _w975, _w976, _w977, _w978, _w979, _w980, _w981, _w982, _w983 : INT;
END_VAR

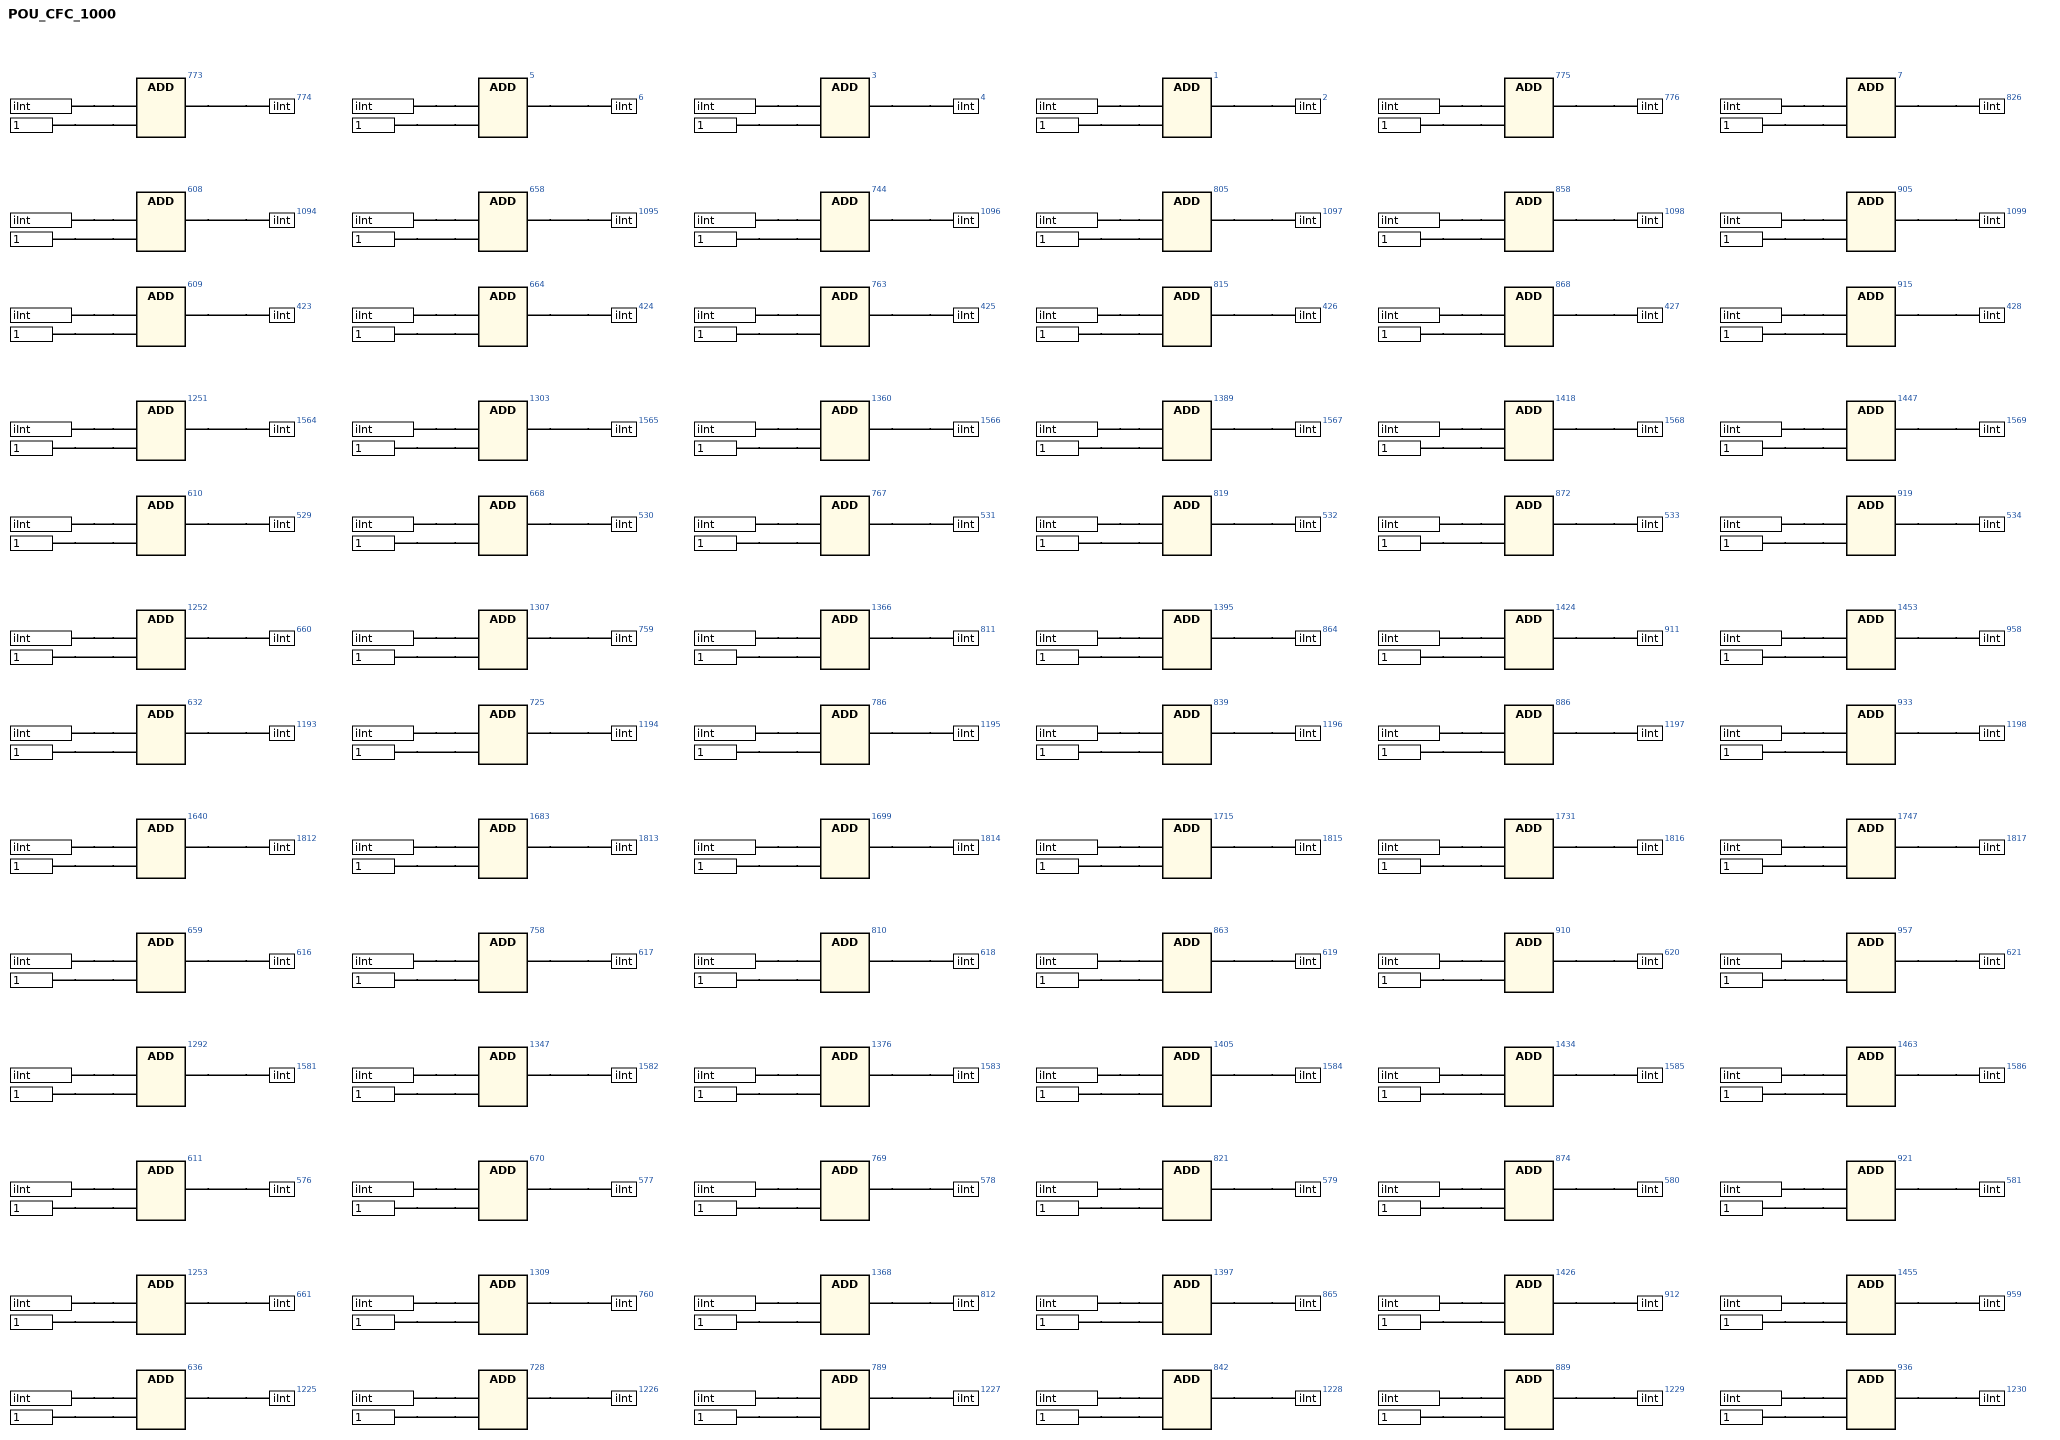
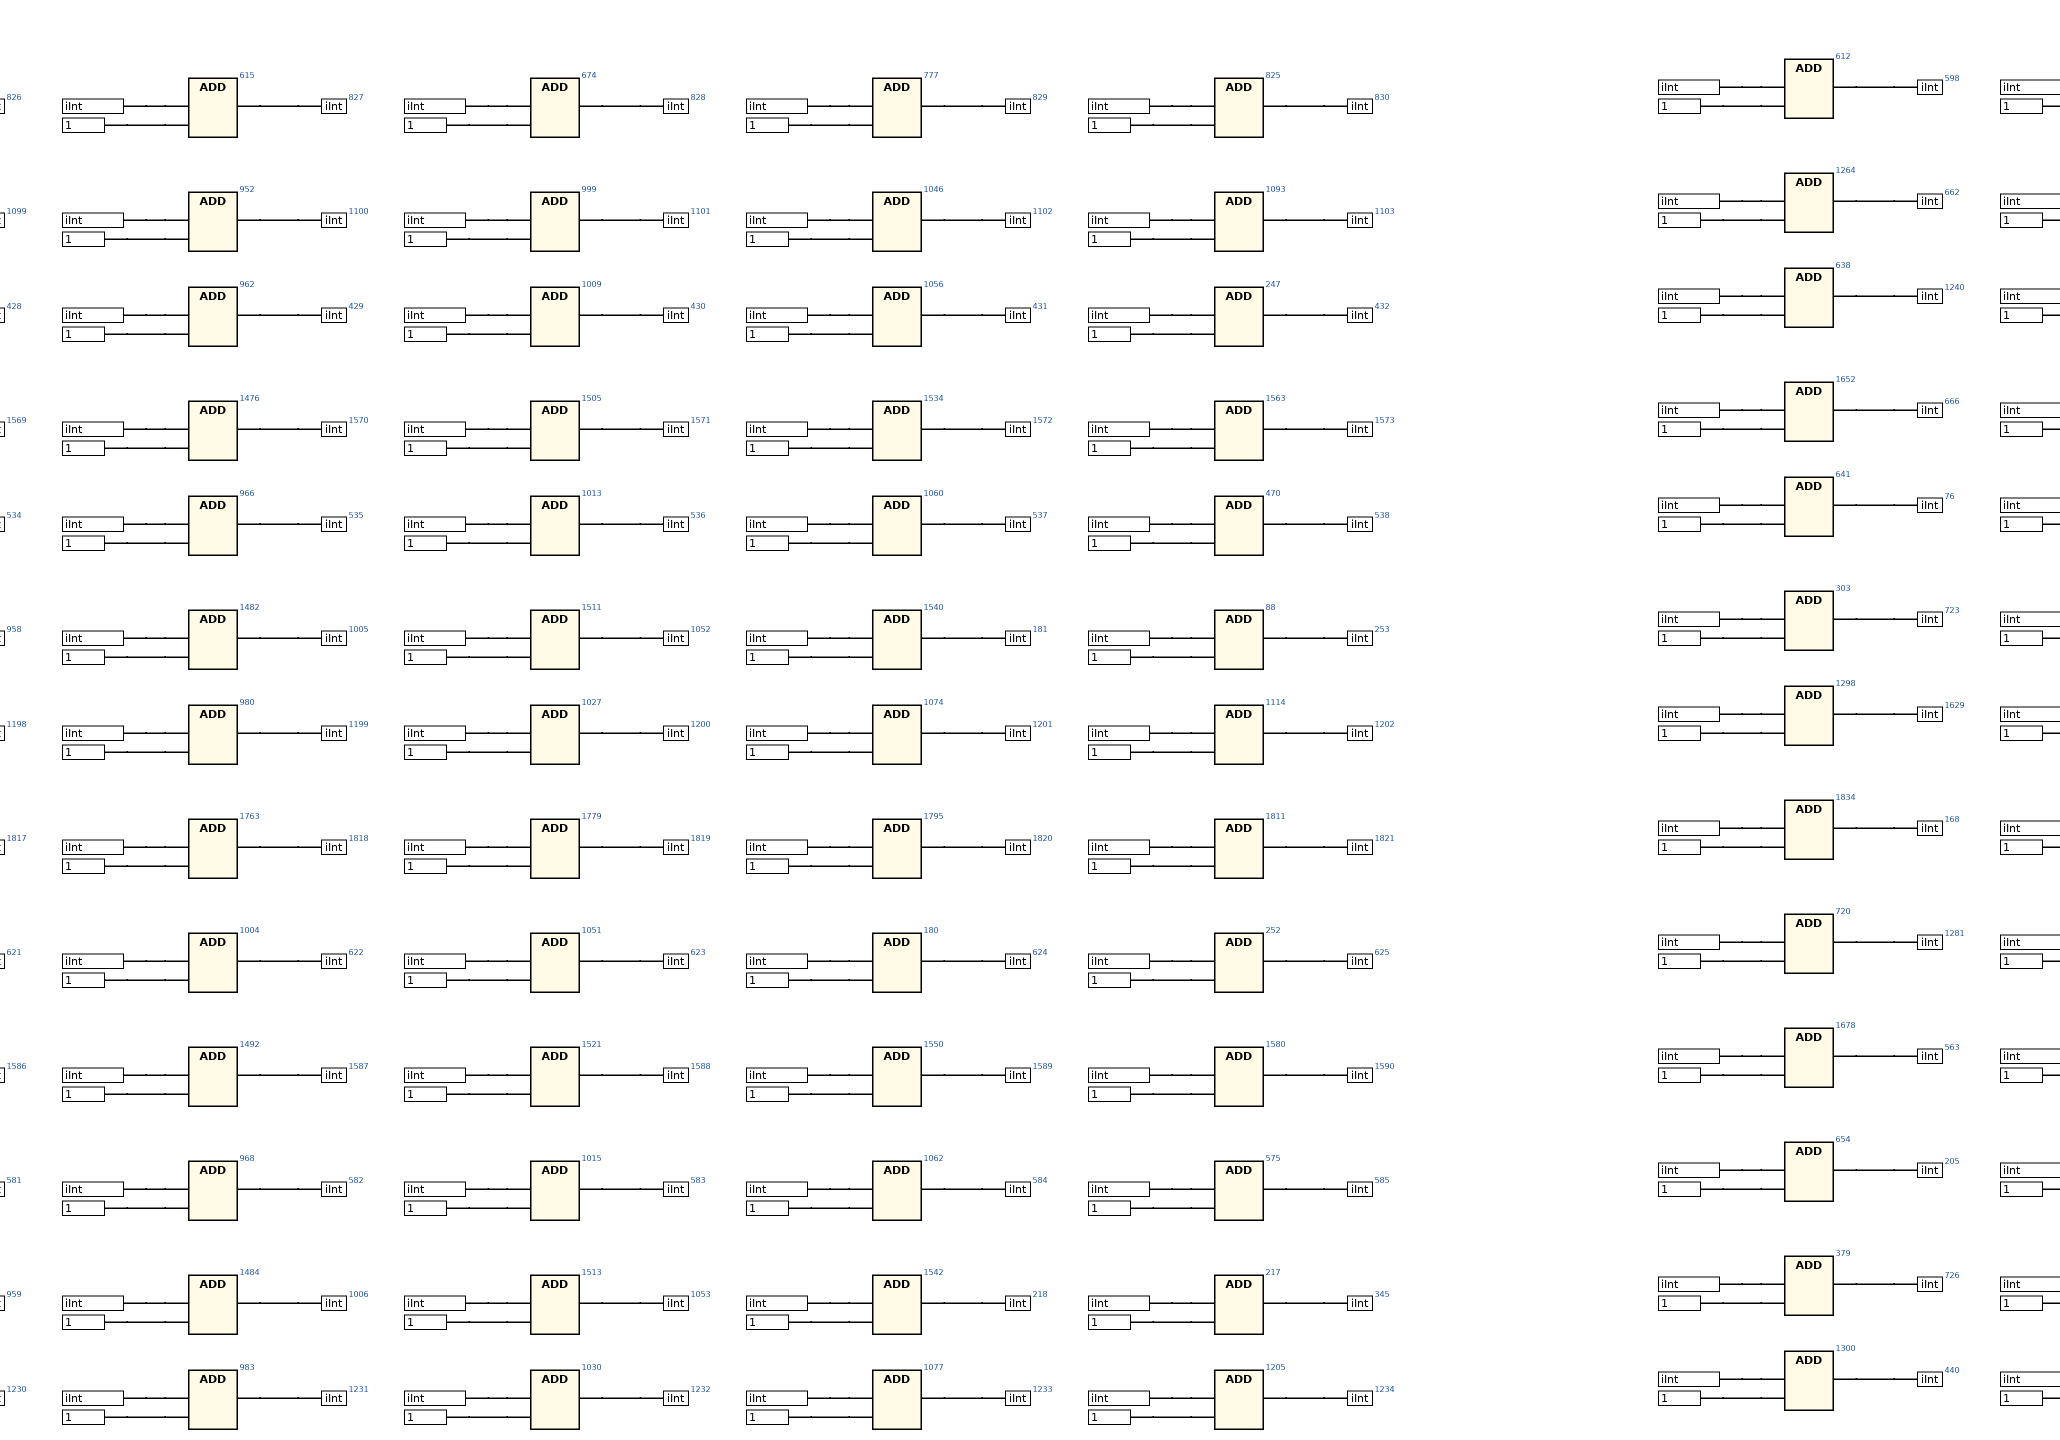
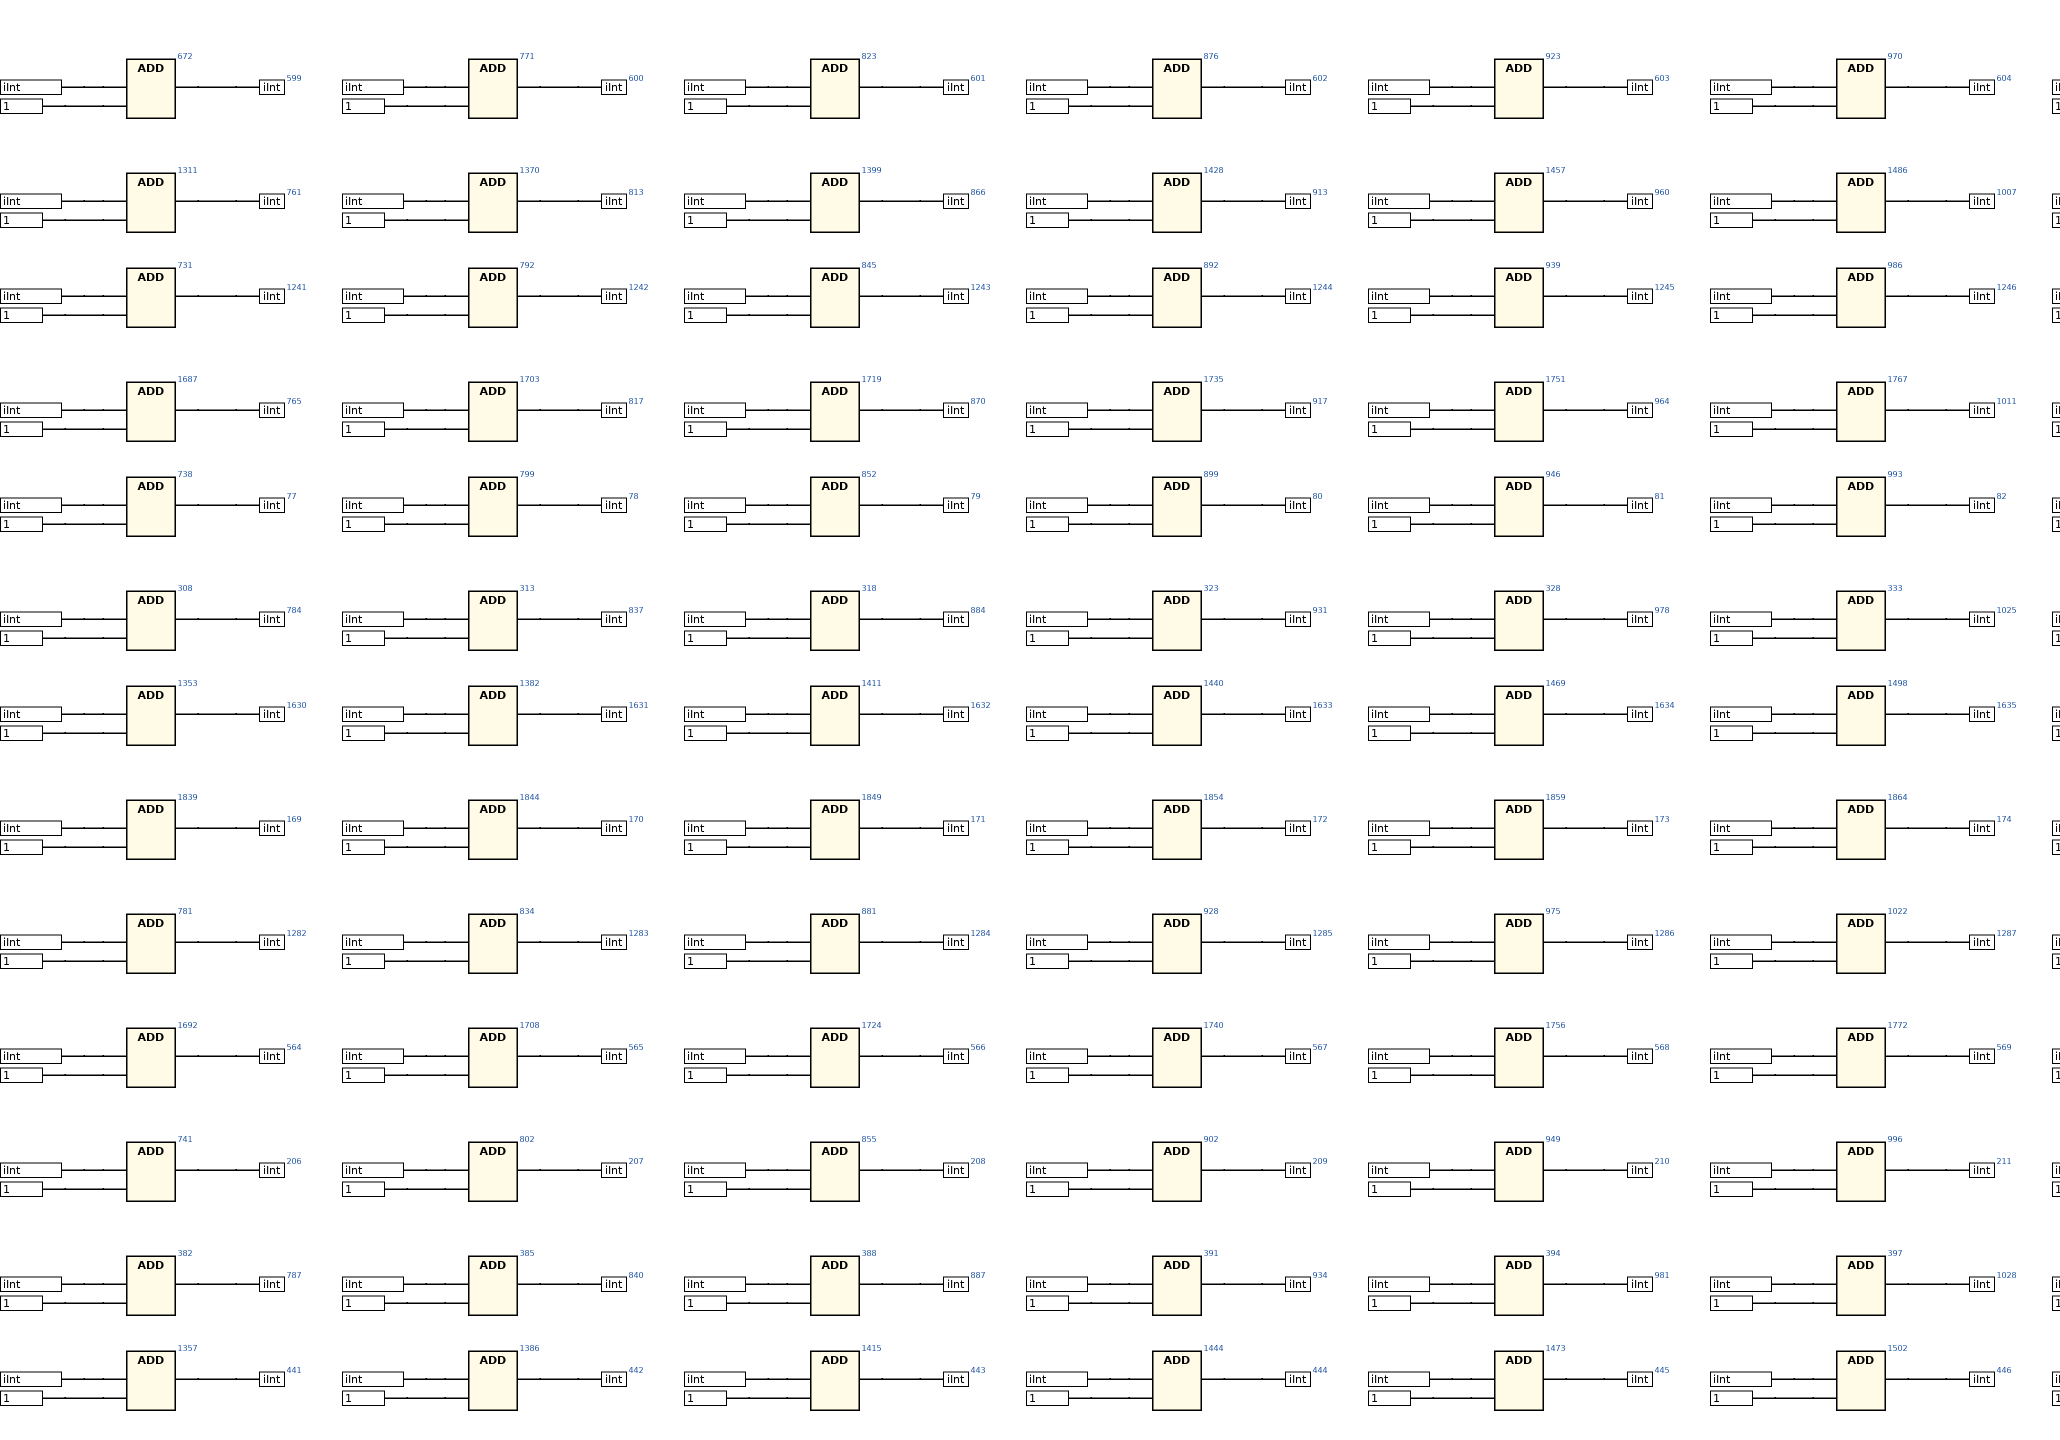
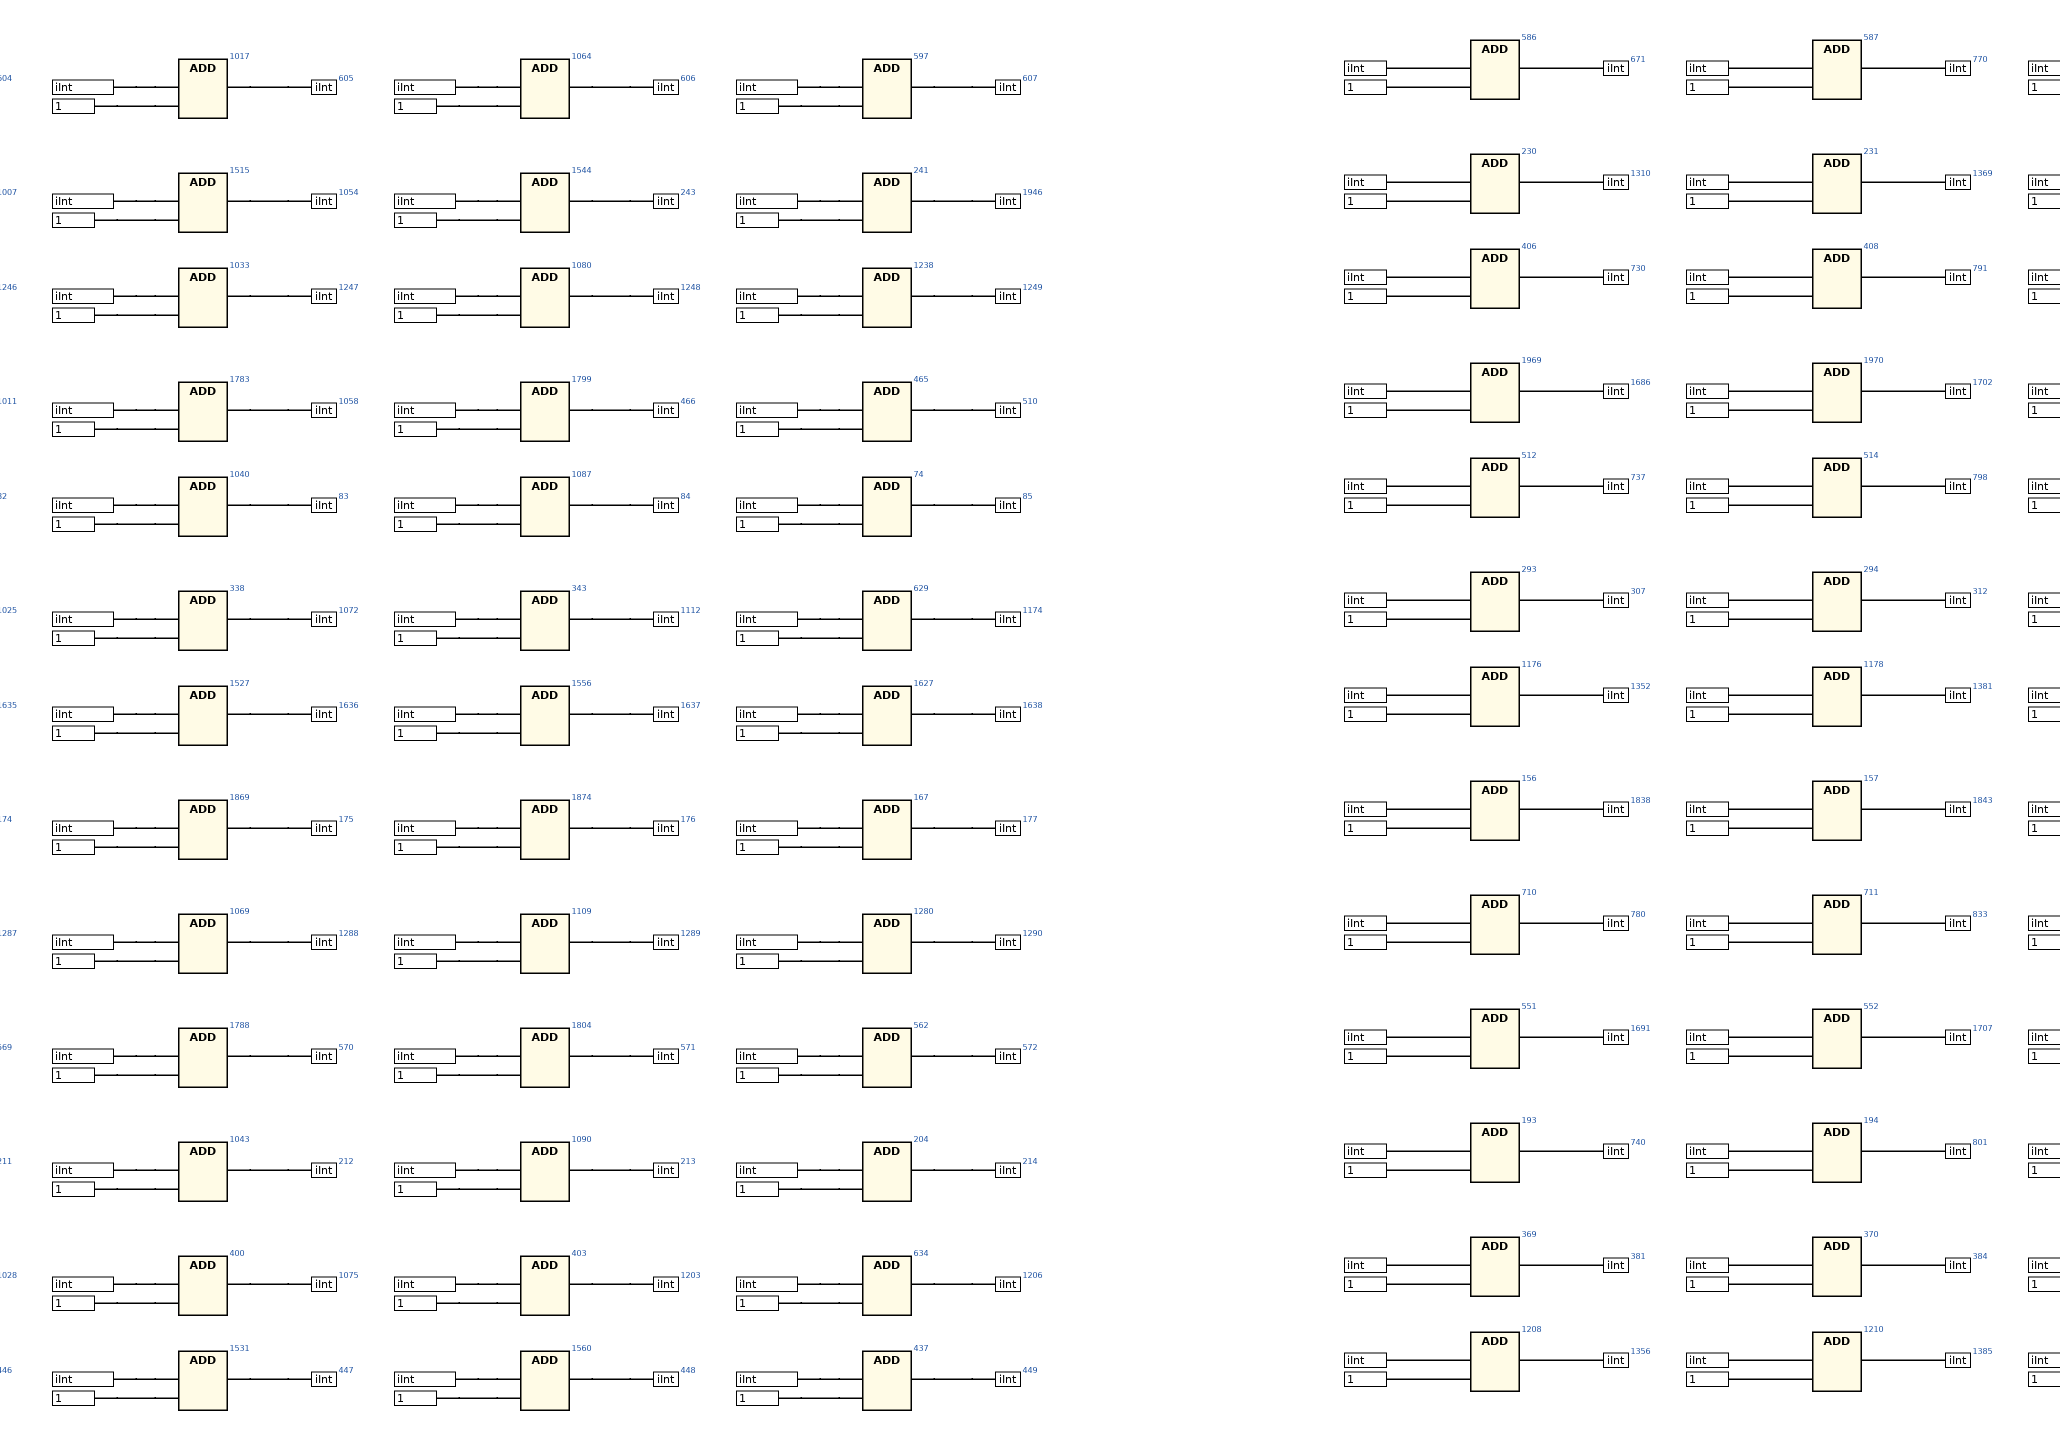
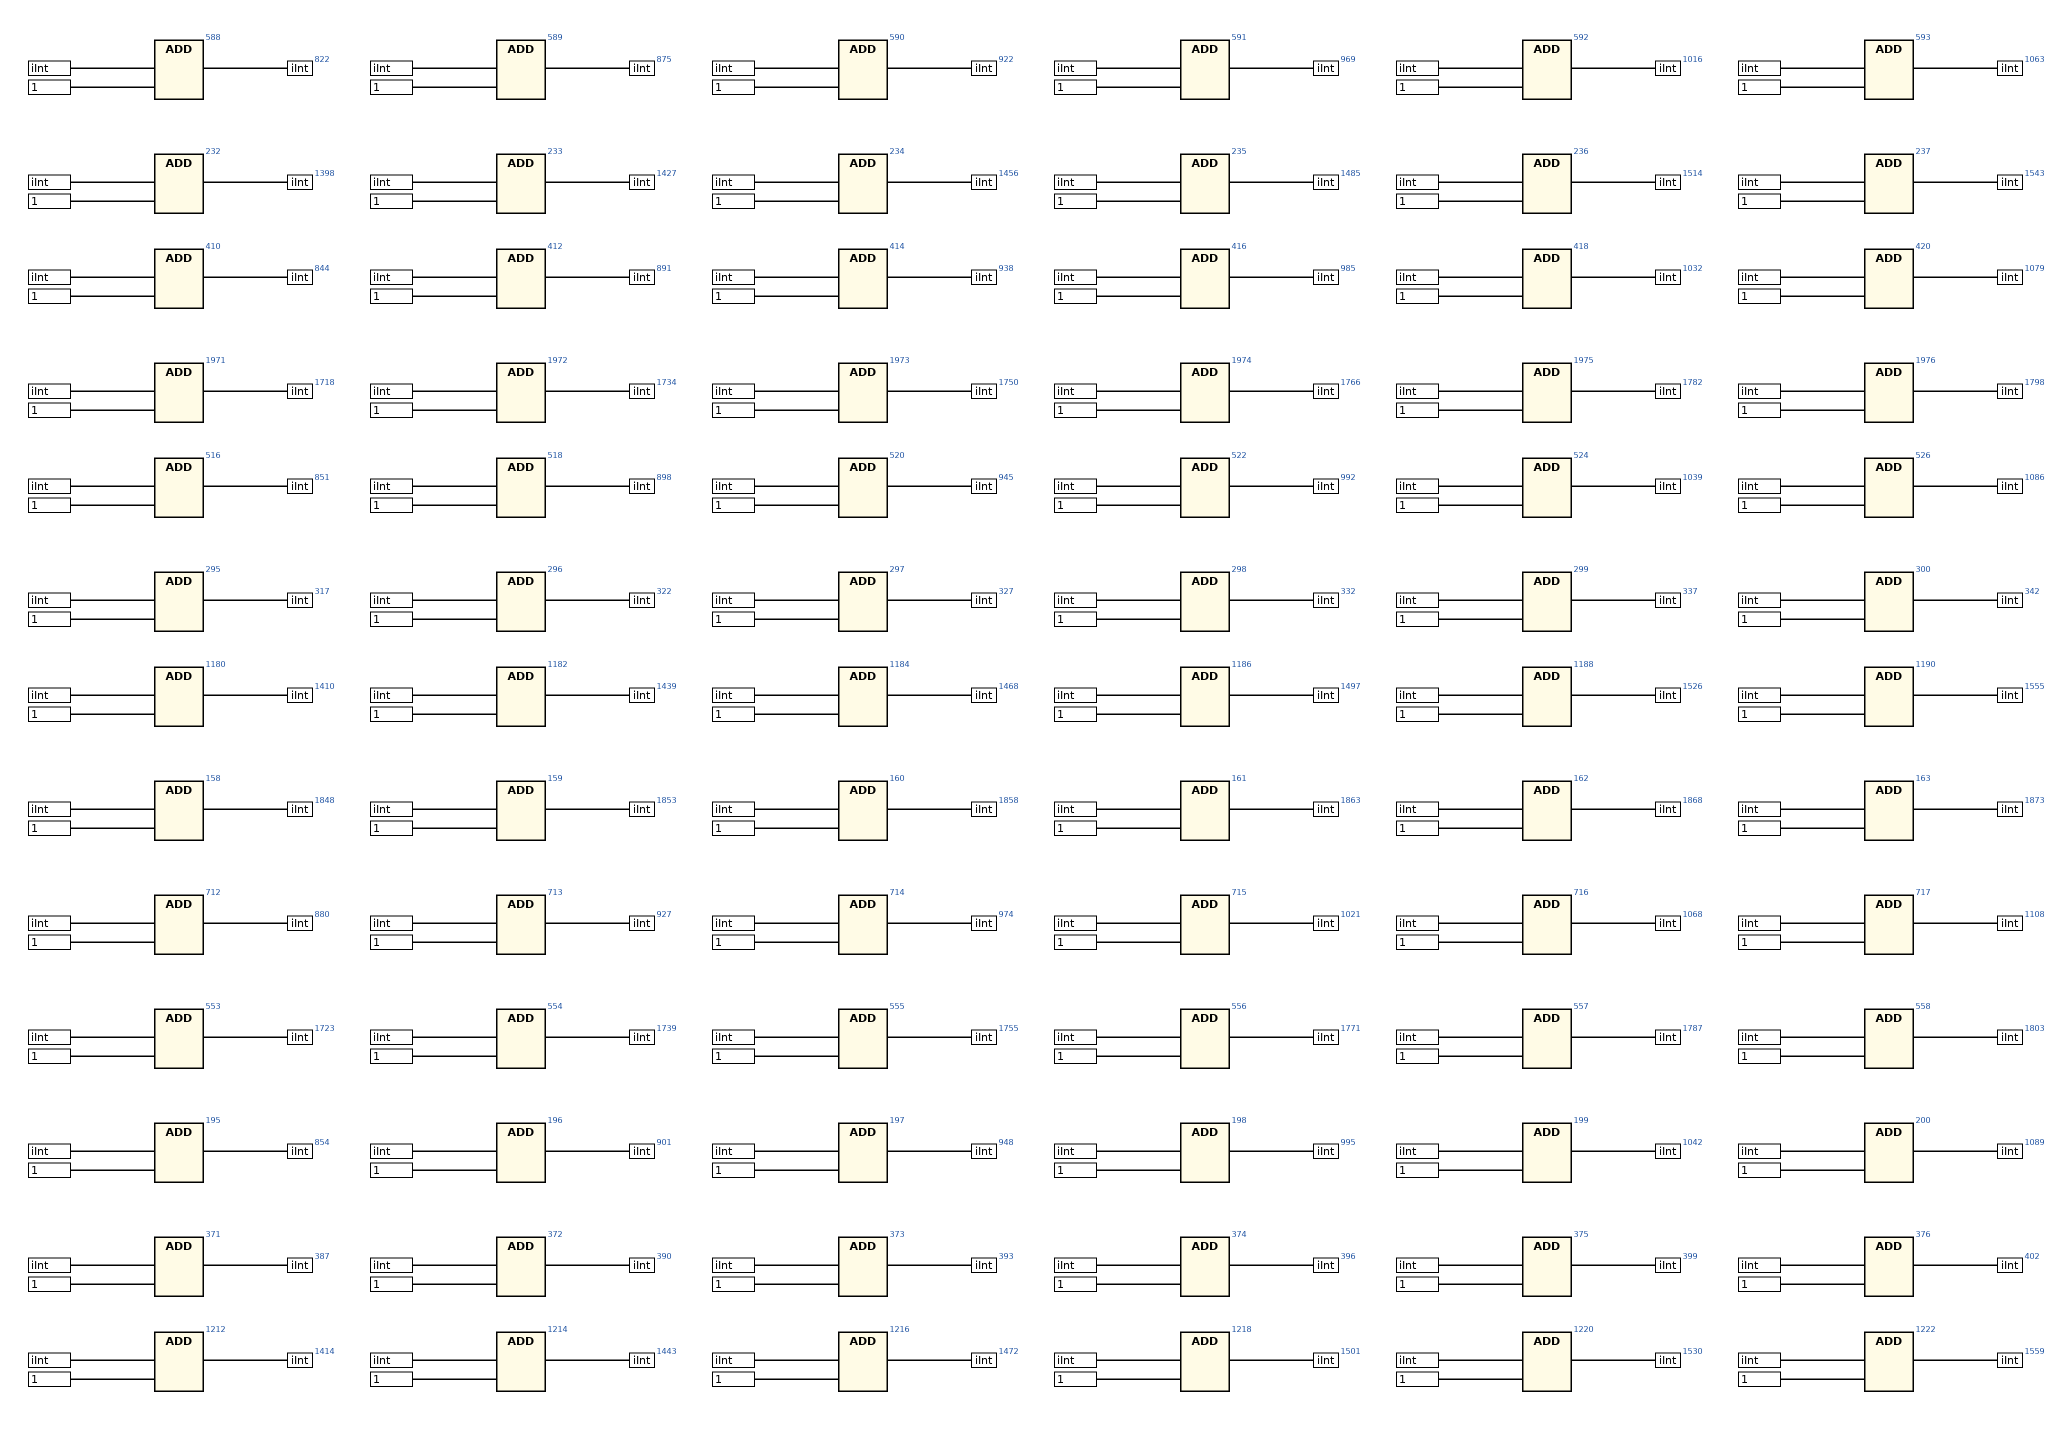
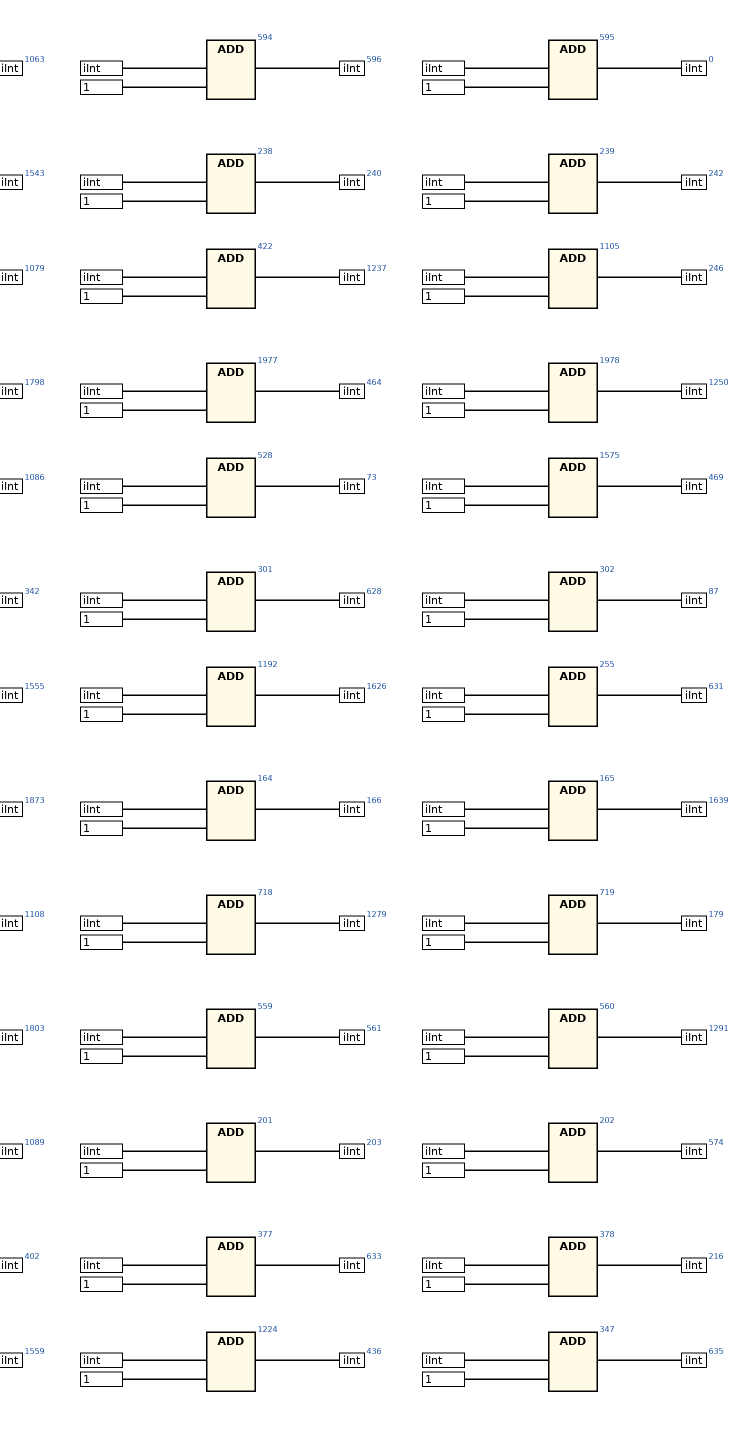
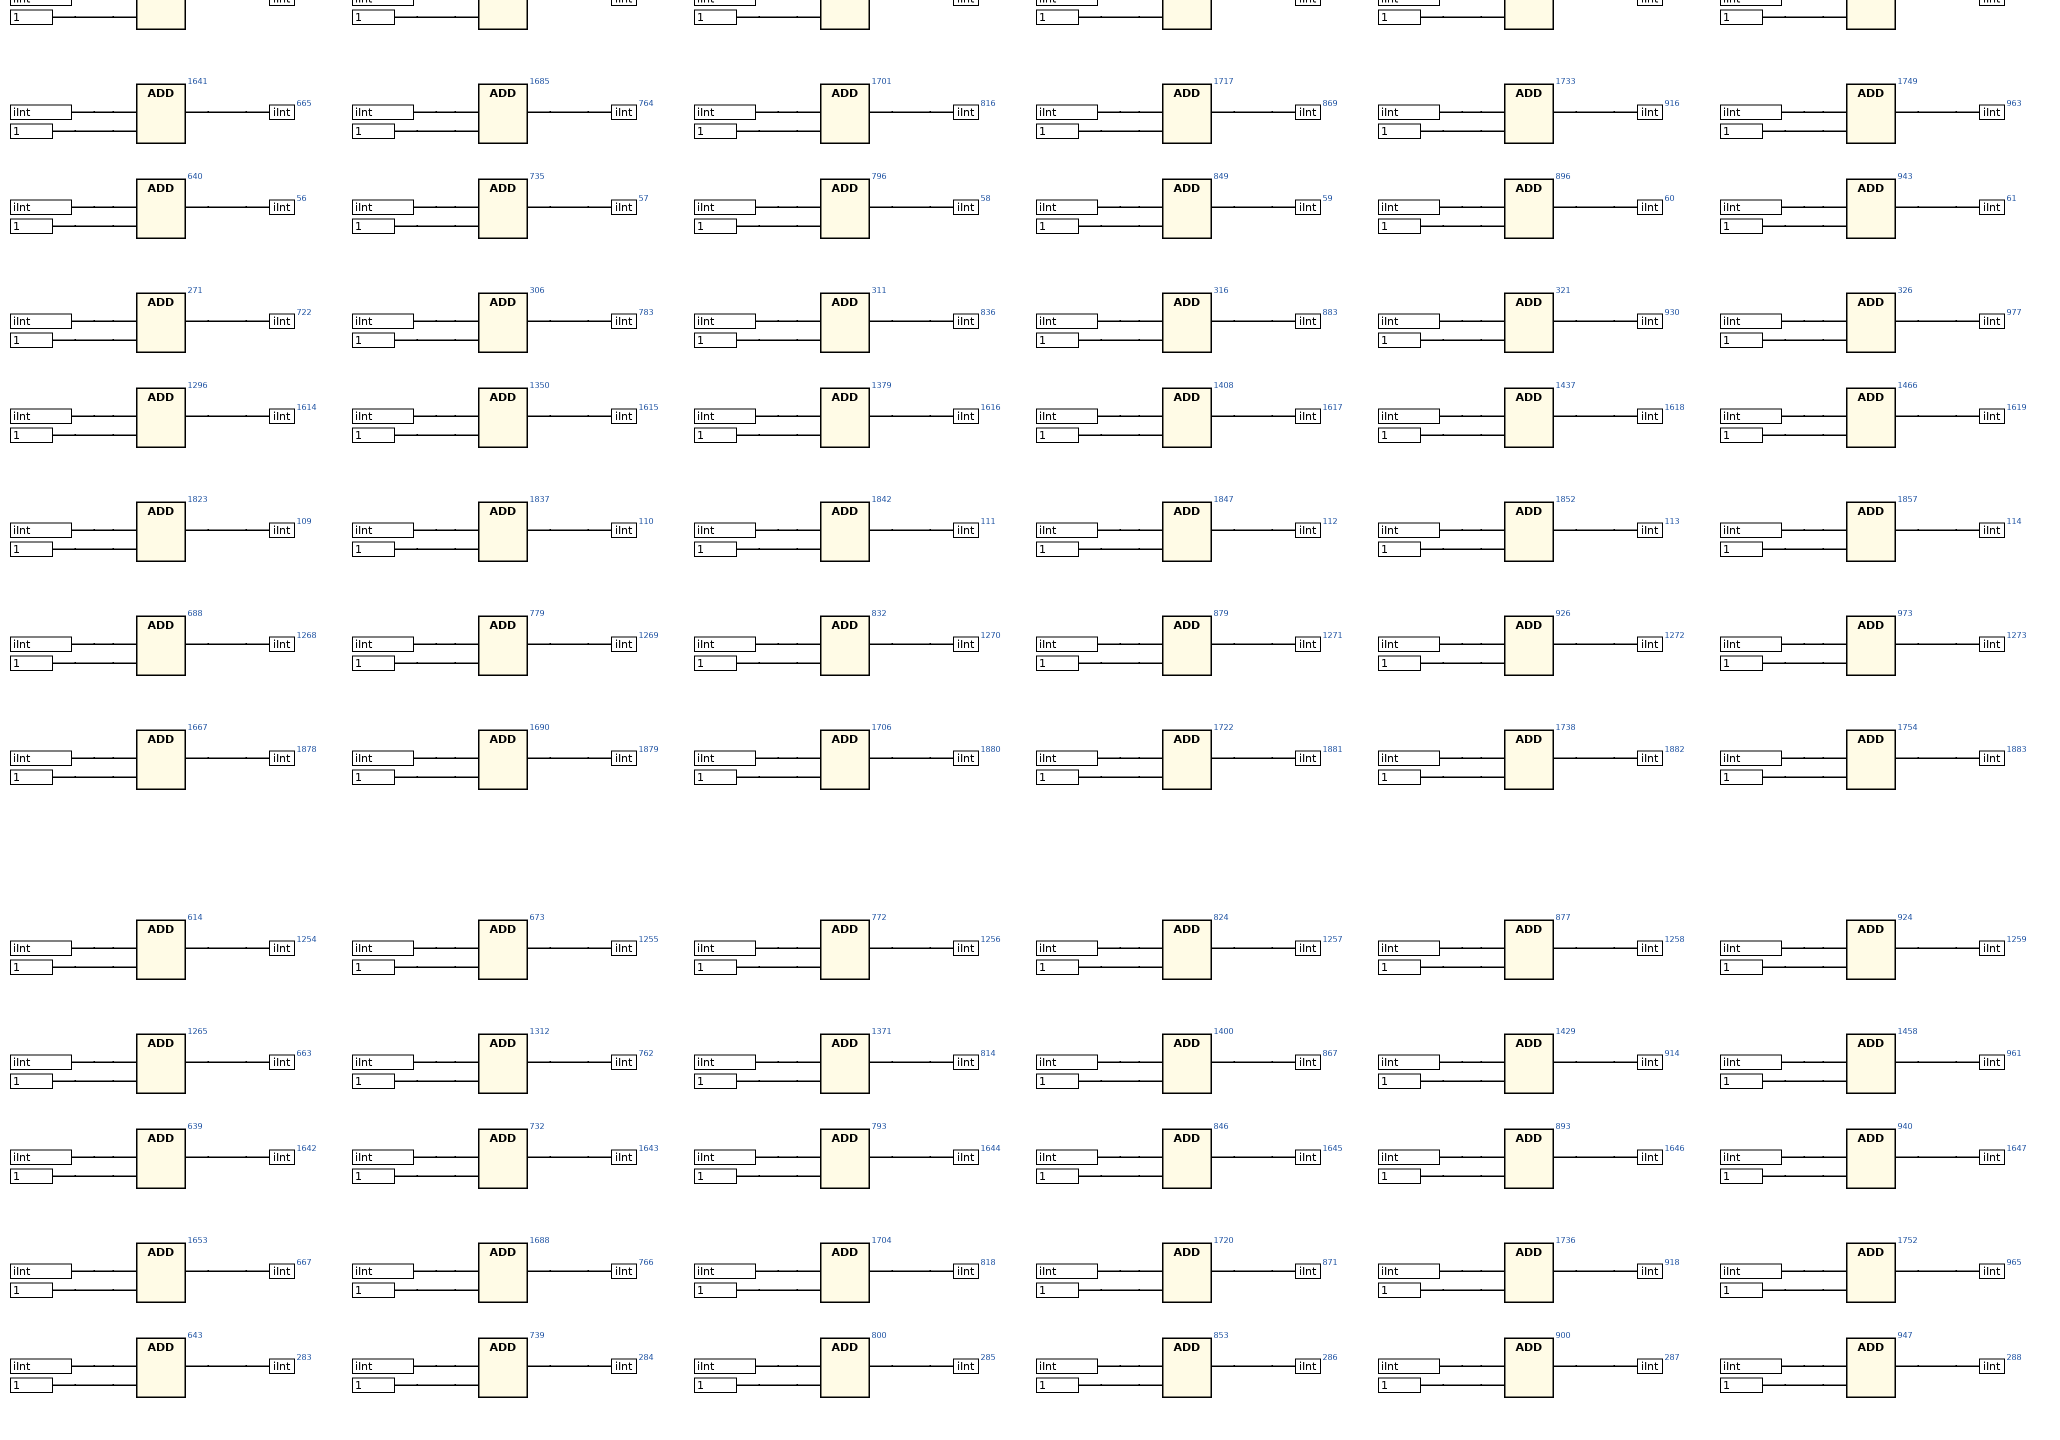
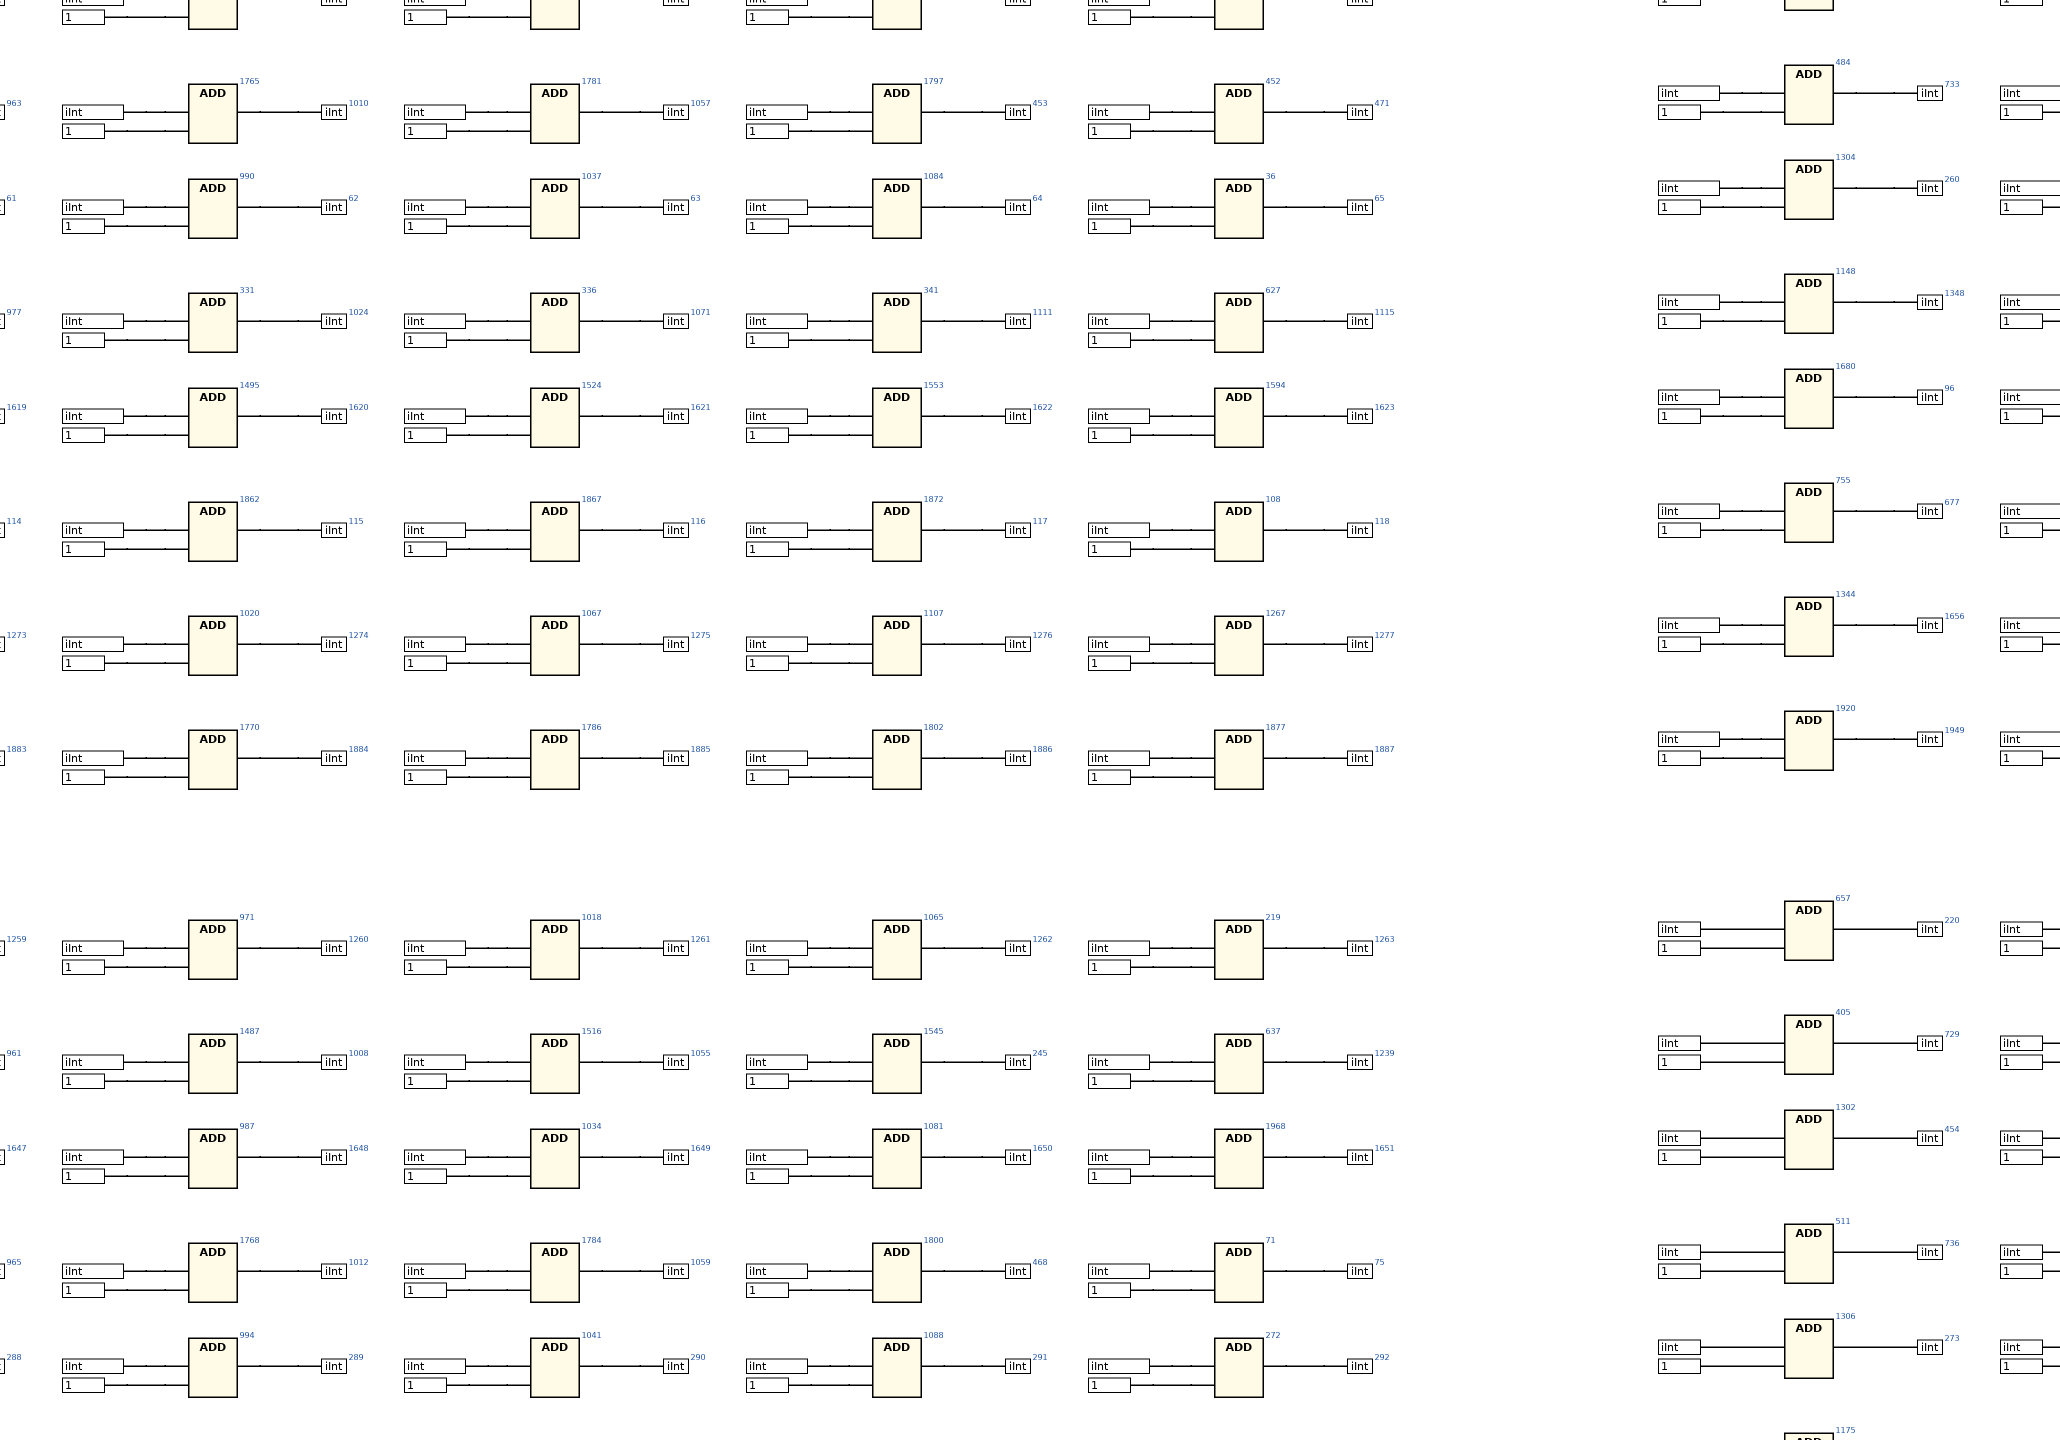
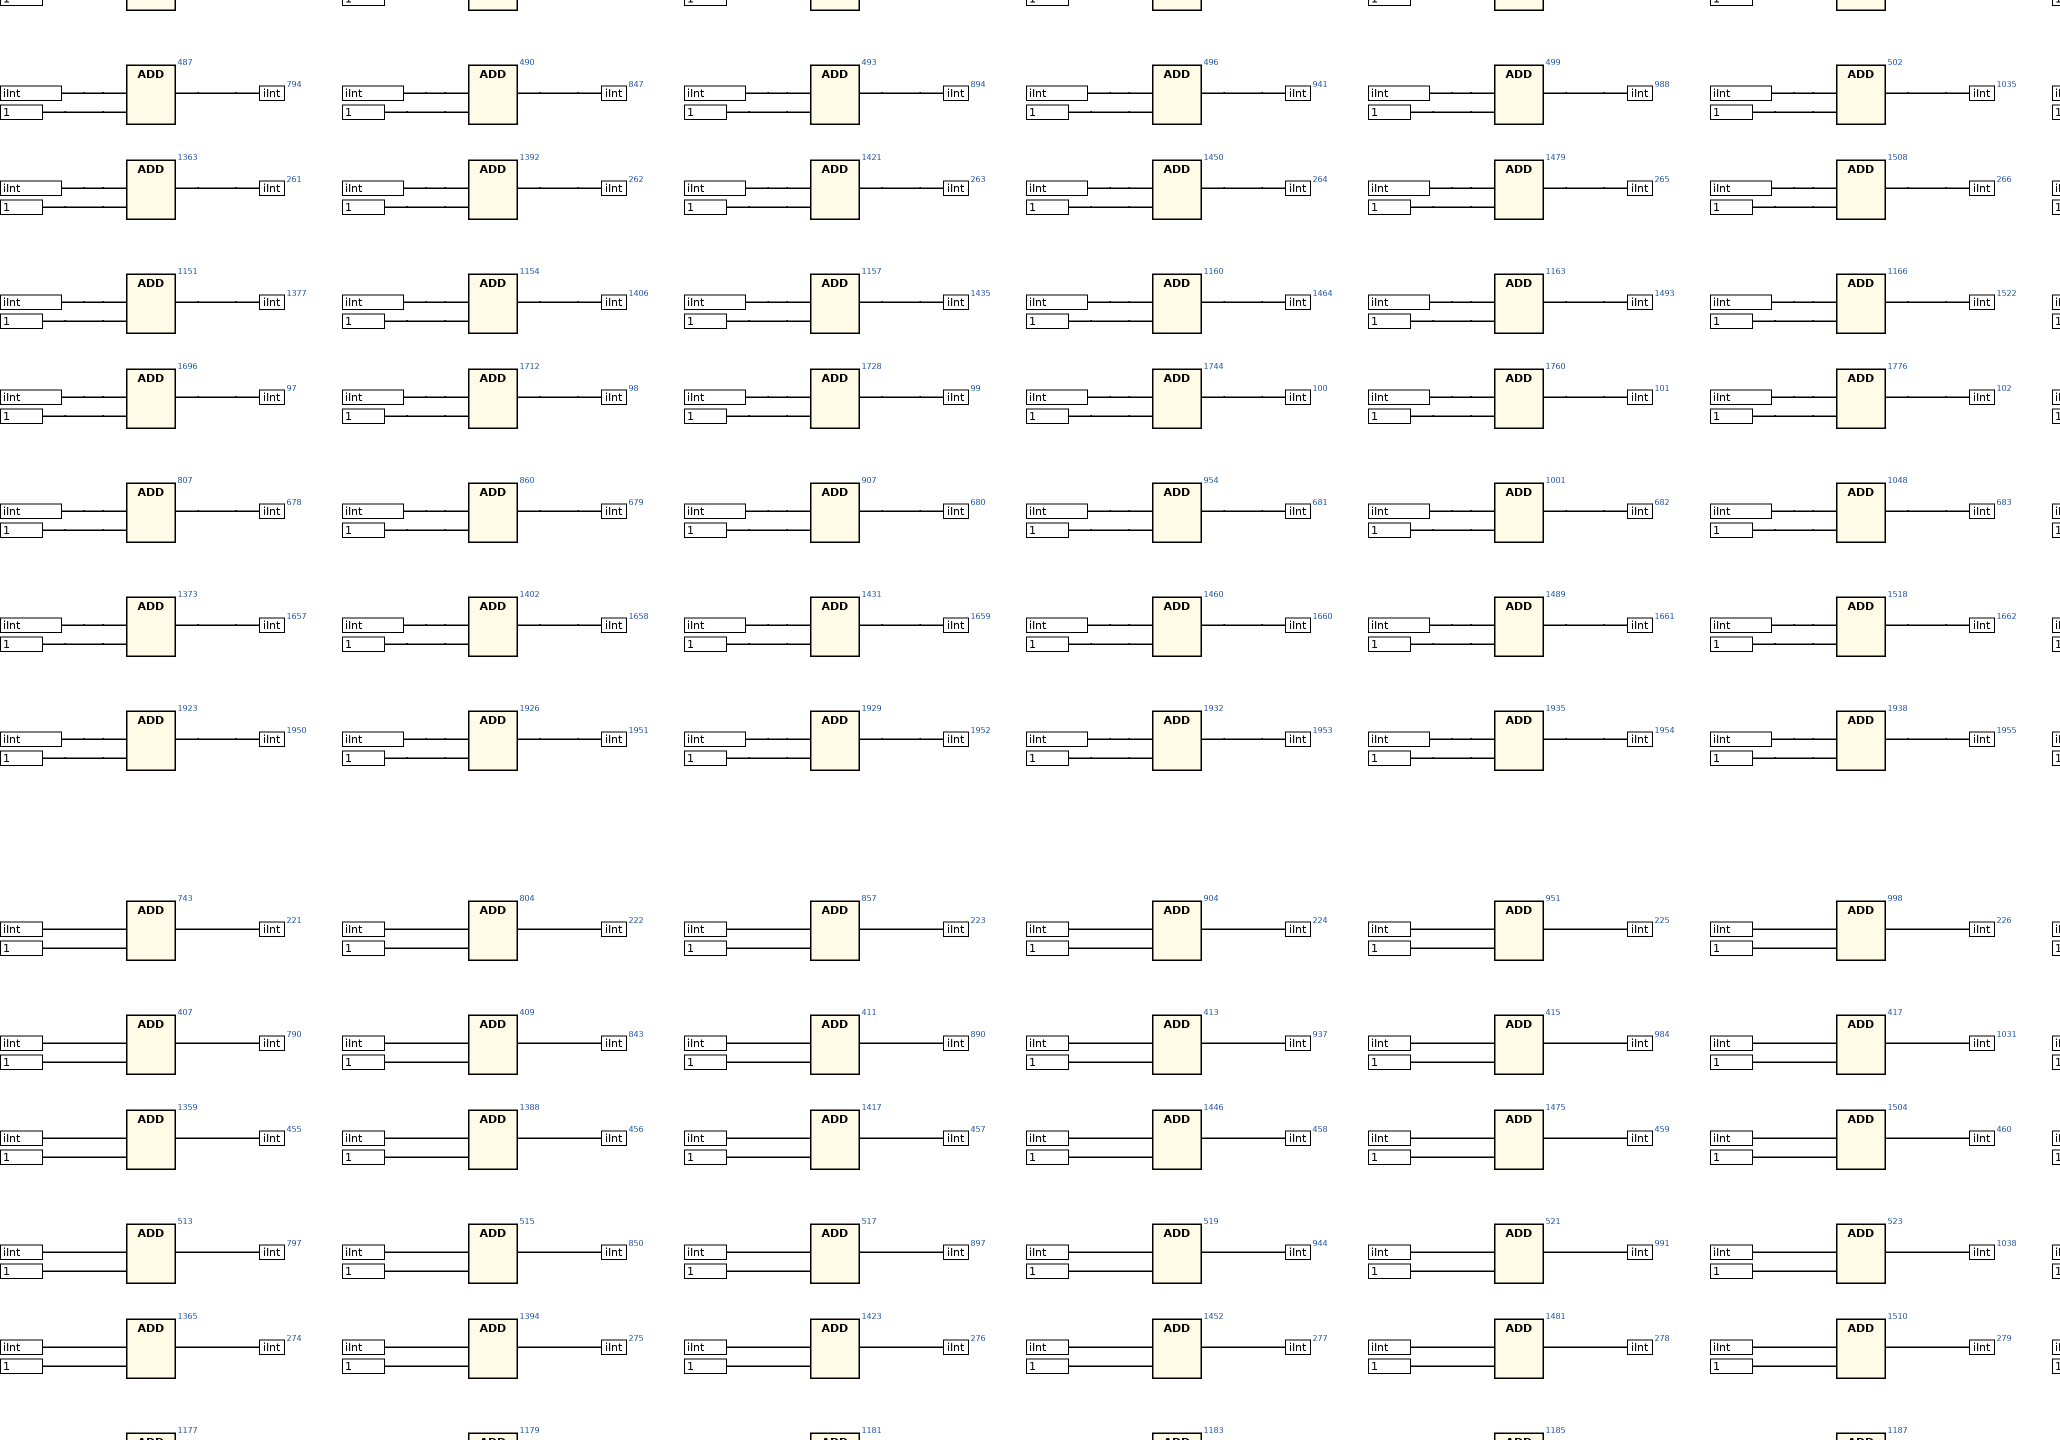
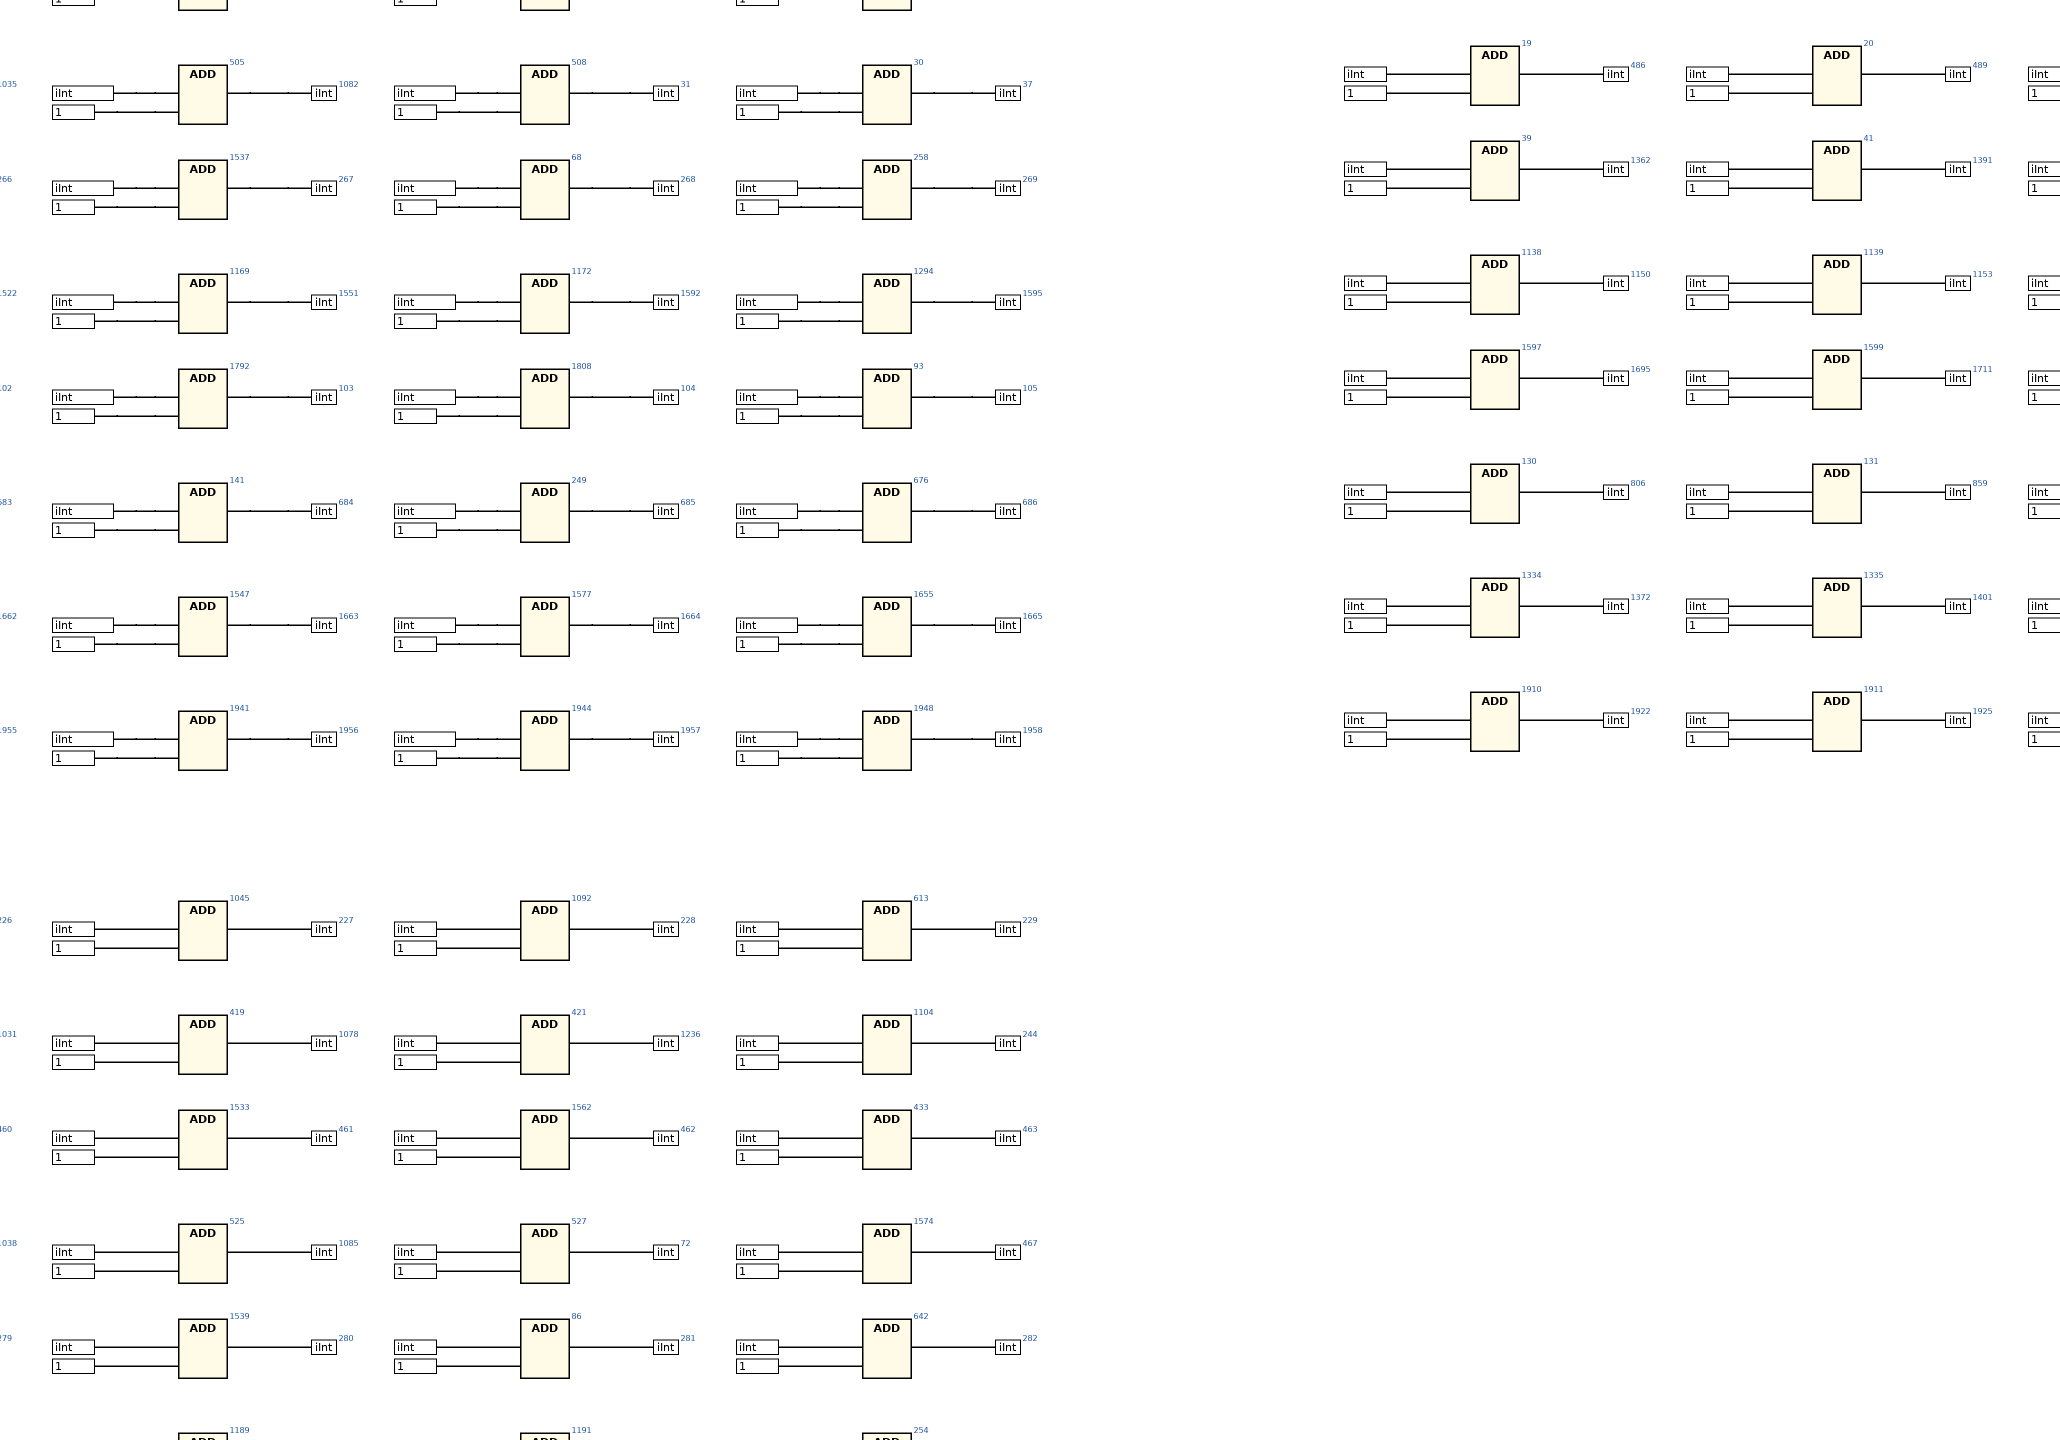
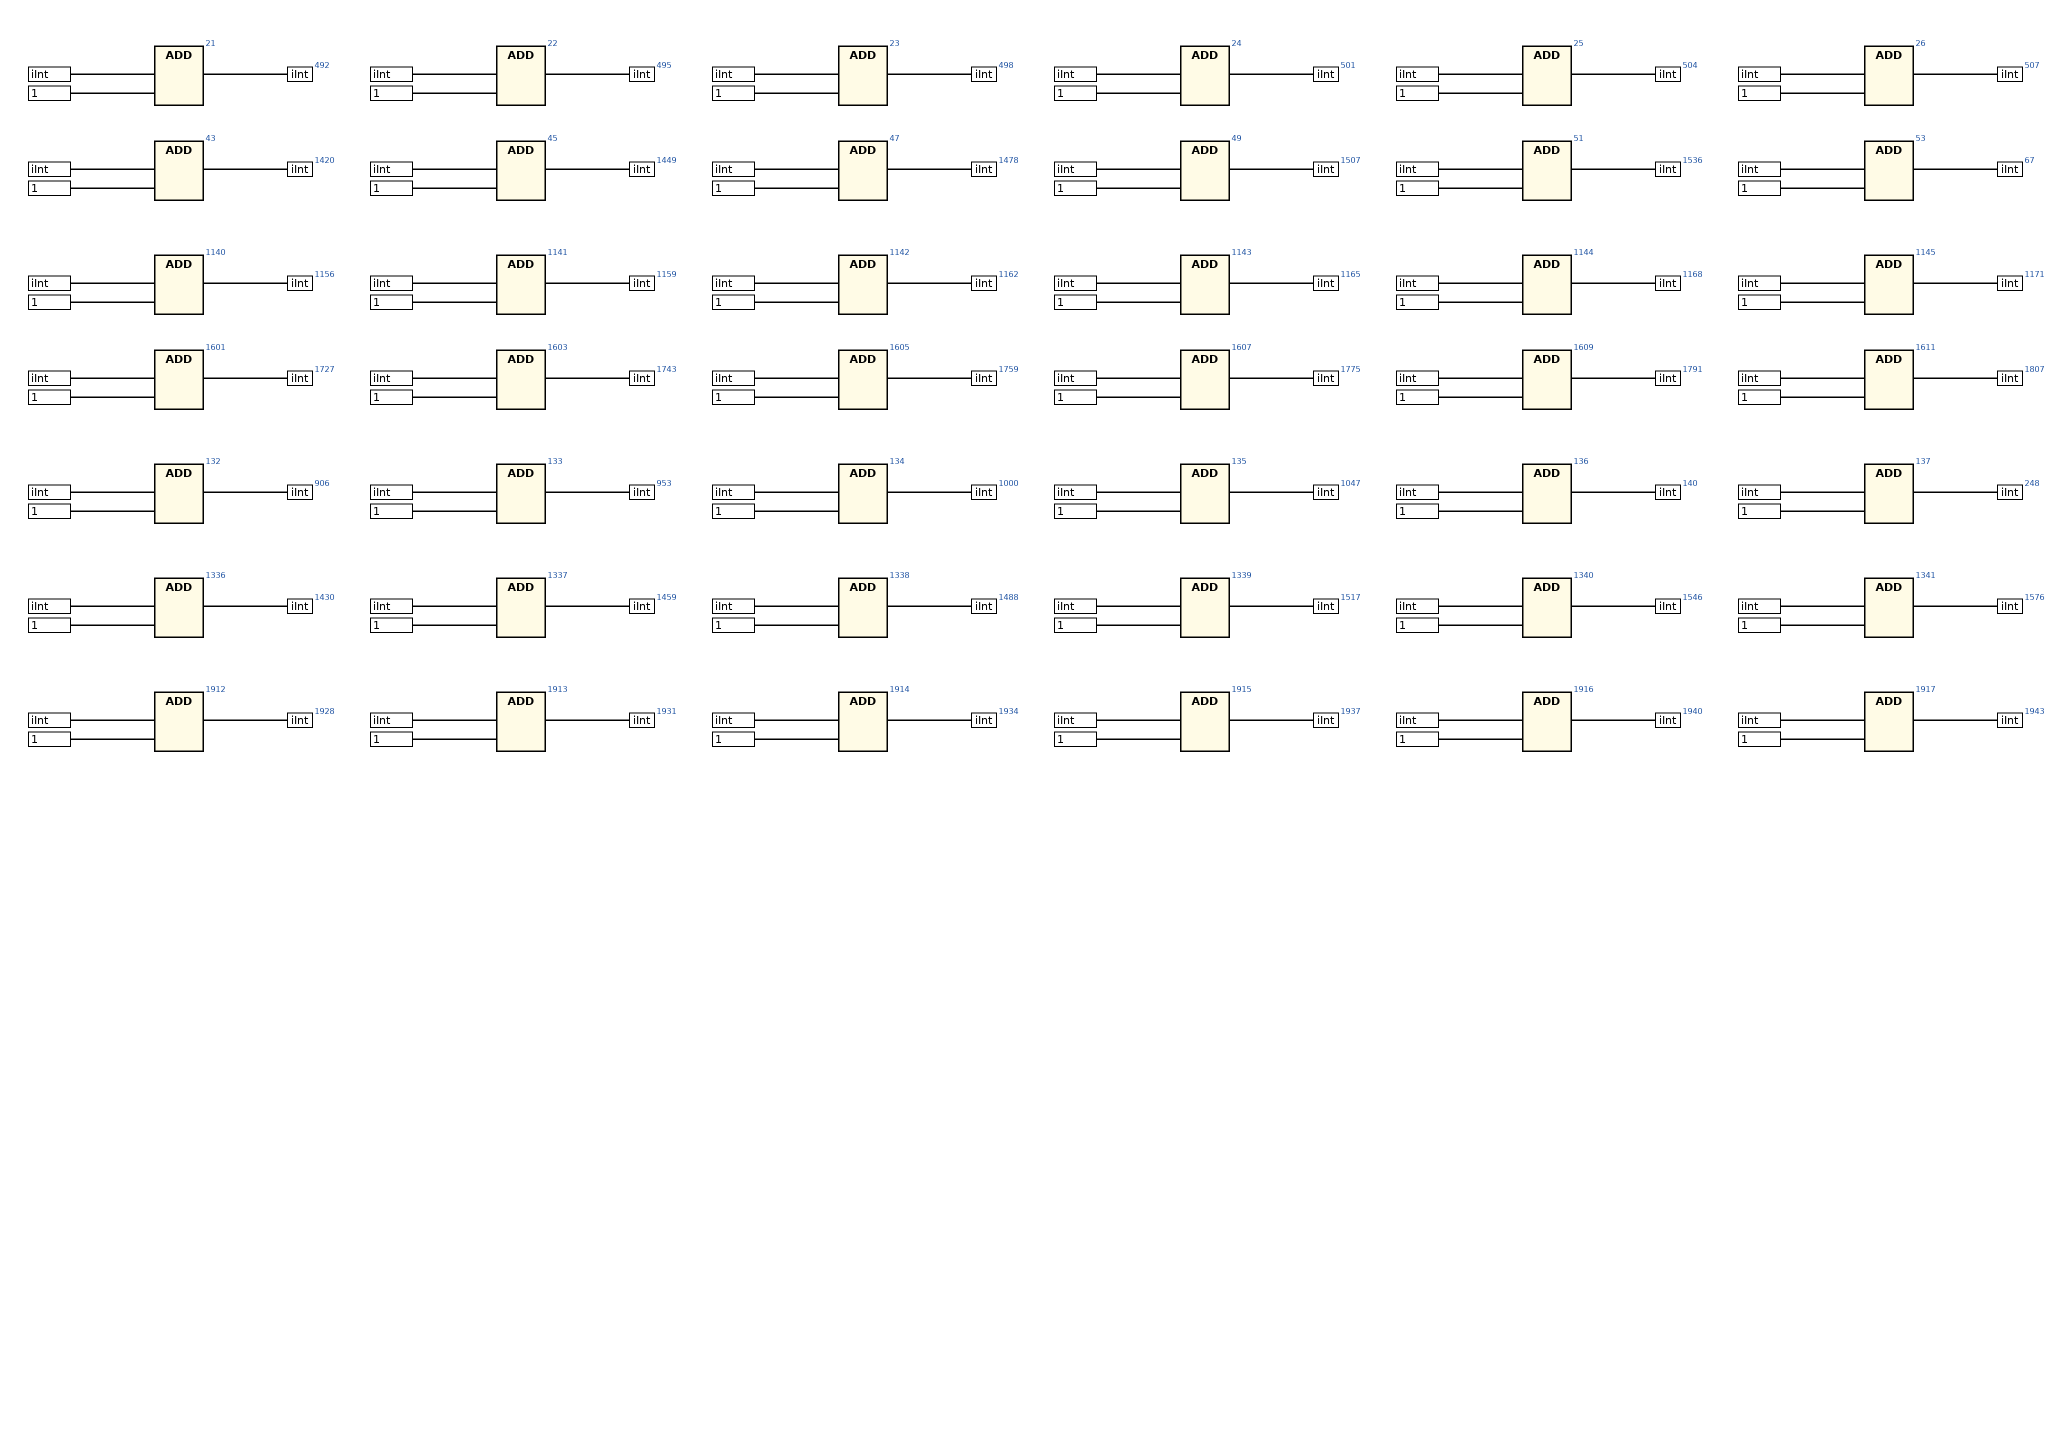
